LIN {X 0,Y 509.786,Z 242.479,A -85,B 0,C 180,E1 -5563.168,E2 -5563.168} C_VEL
LIN {X 0,Y 509.851,Z 242.473,A -85,B 0,C 180,E1 -5565.63,E2 -5565.63} C_VEL
LIN {X 0,Y 509.908,Z 242.464,A -85,B 0,C 180,E1 -5568.87,E2 -5568.87} C_VEL
LIN {X 0,Y 509.872,Z 242.475,A -85,B 0,C 180,E1 -5572.073,E2 -5572.073} C_VEL
LIN {X 0,Y 509.934,Z 242.462,A -85,B 0,C 180,E1 -5574.459,E2 -5574.459} C_VEL
LIN {X 0,Y 510.033,Z 242.455,A -85,B 0,C 180,E1 -5577.626,E2 -5577.626} C_VEL
LIN {X 0,Y 510.023,Z 242.454,A -85,B 0,C 180,E1 -5579.995,E2 -5579.995} C_VEL
LIN {X 0,Y 510.034,Z 242.449,A -85,B 0,C 180,E1 -5582.364,E2 -5582.364} C_VEL
LIN {X 0,Y 509.951,Z 242.467,A -85,B 0,C 180,E1 -5585.531,E2 -5585.531} C_VEL
LIN {X 0,Y 509.905,Z 242.467,A -85,B 0,C 180,E1 -5587.917,E2 -5587.917} C_VEL
LIN {X 0,Y 509.894,Z 242.471,A -85,B 0,C 180,E1 -5591.121,E2 -5591.121} C_VEL
LIN {X 0,Y 509.825,Z 242.474,A -85,B 0,C 180,E1 -5594.361,E2 -5594.361} C_VEL
LIN {X 0,Y 509.844,Z 242.475,A -85,B 0,C 180,E1 -5596.821,E2 -5596.821} C_VEL
LIN {X 0,Y 509.889,Z 242.466,A -85,B 0,C 180,E1 -5600.15,E2 -5600.15} C_VEL
LIN {X 0,Y 509.793,Z 242.48,A -85,B 0,C 180,E1 -5603.559,E2 -5603.559} C_VEL
LIN {X 0,Y 509.88,Z 242.469,A -85,B 0,C 180,E1 -5606.373,E2 -5606.373} C_VEL
LIN {X 0,Y 509.843,Z 242.481,A -85,B 0,C 180,E1 -5608.839,E2 -5608.839} C_VEL
LIN {X 0,Y 509.783,Z 242.48,A -85,B 0,C 180,E1 -5611.585,E2 -5611.585} C_VEL
LIN {X 0,Y 509.815,Z 242.48,A -85,B 0,C 180,E1 -5614.408,E2 -5614.408} C_VEL
LIN {X 0,Y 509.777,Z 242.481,A -85,B 0,C 180,E1 -5617.336,E2 -5617.336} C_VEL
LIN {X 0,Y 509.798,Z 242.485,A -85,B 0,C 180,E1 -5620.377,E2 -5620.377} C_VEL
LIN {X 0,Y 509.793,Z 242.479,A -85,B 0,C 180,E1 -5623.06,E2 -5623.06} C_VEL
LIN {X 0,Y 509.781,Z 242.482,A -85,B 0,C 180,E1 -5625.788,E2 -5625.788} C_VEL
LIN {X 0,Y 509.814,Z 242.479,A -85,B 0,C 180,E1 -5628.571,E2 -5628.571} C_VEL
LIN {X 0,Y 509.805,Z 242.479,A -85,B 0,C 180,E1 -5631.659,E2 -5631.659} C_VEL
LIN {X 0,Y 509.777,Z 242.483,A -85,B 0,C 180,E1 -5633.695,E2 -5633.695} C_VEL
LIN {X 0,Y 509.109,Z 242.568,A -85,B 0,C 180,E1 -5634.355,E2 -5634.355} C_VEL
LIN {X 0,Y 506.293,Z 242.916,A -85,B 0,C 180,E1 -5635.427,E2 -5635.427} C_VEL
LIN {X 0,Y 503.902,Z 243.217,A -85,B 0,C 180,E1 -5636.29,E2 -5636.29} C_VEL
LIN {X 0,Y 502.854,Z 243.343,A -85,B 0,C 180,E1 -5636.956,E2 -5636.956} C_VEL
LIN {X 0,Y 502.756,Z 243.355,A -85,B 0,C 180,E1 -5637.182,E2 -5637.182} C_VEL
LIN {X 0,Y 502.773,Z 243.359,A -85,B 0,C 180,E1 -5640.058,E2 -5640.058} C_VEL
LIN {X 0,Y 502.775,Z 243.353,A -85,B 0,C 180,E1 -5642.53,E2 -5642.53} C_VEL
LIN {X 0,Y 502.782,Z 243.354,A -85,B 0,C 180,E1 -5645.292,E2 -5645.292} C_VEL
LIN {X 0,Y 502.757,Z 243.361,A -85,B 0,C 180,E1 -5647.826,E2 -5647.826} C_VEL
LIN {X 0,Y 502.762,Z 243.354,A -85,B 0,C 180,E1 -5650.398,E2 -5650.398} C_VEL
LIN {X 0,Y 502.784,Z 243.355,A -85,B 0,C 180,E1 -5652.93,E2 -5652.93} C_VEL
LIN {X 0,Y 502.797,Z 243.359,A -85,B 0,C 180,E1 -5655.428,E2 -5655.428} C_VEL
LIN {X 0,Y 502.831,Z 243.349,A -85,B 0,C 180,E1 -5658.716,E2 -5658.716} C_VEL
LIN {X 0,Y 502.851,Z 243.346,A -85,B 0,C 180,E1 -5661.966,E2 -5661.966} C_VEL
LIN {X 0,Y 502.899,Z 243.34,A -85,B 0,C 180,E1 -5664.386,E2 -5664.386} C_VEL
LIN {X 0,Y 502.96,Z 243.333,A -85,B 0,C 180,E1 -5667.598,E2 -5667.598} C_VEL
LIN {X 0,Y 502.955,Z 243.333,A -85,B 0,C 180,E1 -5670,E2 -5670} C_VEL
LIN {X 0,Y 502.96,Z 243.333,A -85,B 0,C 180,E1 -5672.402,E2 -5672.402} C_VEL
LIN {X 0,Y 502.899,Z 243.34,A -85,B 0,C 180,E1 -5675.614,E2 -5675.614} C_VEL
LIN {X 0,Y 502.851,Z 243.346,A -85,B 0,C 180,E1 -5678.034,E2 -5678.034} C_VEL
LIN {X 0,Y 502.831,Z 243.349,A -85,B 0,C 180,E1 -5681.284,E2 -5681.284} C_VEL
LIN {X 0,Y 502.797,Z 243.359,A -85,B 0,C 180,E1 -5684.572,E2 -5684.572} C_VEL
LIN {X 0,Y 502.813,Z 243.352,A -85,B 0,C 180,E1 -5687.908,E2 -5687.908} C_VEL
LIN {X 0,Y 502.766,Z 243.36,A -85,B 0,C 180,E1 -5690.539,E2 -5690.539} C_VEL
LIN {X 0,Y 502.76,Z 243.355,A -85,B 0,C 180,E1 -5693.042,E2 -5693.042} C_VEL
LIN {X 0,Y 502.792,Z 243.352,A -85,B 0,C 180,E1 -5695.678,E2 -5695.678} C_VEL
LIN {X 0,Y 502.782,Z 243.357,A -85,B 0,C 180,E1 -5698.376,E2 -5698.376} C_VEL
LIN {X 0,Y 502.745,Z 243.358,A -85,B 0,C 180,E1 -5701.504,E2 -5701.504} C_VEL
LIN {X 0,Y 502.75,Z 243.358,A -85,B 0,C 180,E1 -5704.448,E2 -5704.448} C_VEL
LIN {X 0,Y 502.726,Z 243.359,A -85,B 0,C 180,E1 -5707.182,E2 -5707.182} C_VEL
LIN {X 0,Y 502.774,Z 243.358,A -85,B 0,C 180,E1 -5710.016,E2 -5710.016} C_VEL
LIN {X 0,Y 502.779,Z 243.354,A -85,B 0,C 180,E1 -5712.207,E2 -5712.207} C_VEL
LIN {X 0,Y 502.753,Z 243.361,A -85,B 0,C 180,E1 -5715.473,E2 -5715.473} C_VEL
LIN {X 0,Y 502.784,Z 243.356,A -85,B 0,C 180,E1 -5717.869,E2 -5717.869} C_VEL
LIN {X 0,Y 502.758,Z 243.357,A -85,B 0,C 180,E1 -5721.029,E2 -5721.029} C_VEL
LIN {X 0,Y 502.745,Z 243.356,A -85,B 0,C 180,E1 -5724.172,E2 -5724.172} C_VEL
LIN {X 0,Y 502.795,Z 243.354,A -85,B 0,C 180,E1 -5726.998,E2 -5726.998} C_VEL
LIN {X 0,Y 502.78,Z 243.352,A -85,B 0,C 180,E1 -5730.07,E2 -5730.07} C_VEL
LIN {X 0,Y 502.802,Z 243.35,A -85,B 0,C 180,E1 -5732.538,E2 -5732.538} C_VEL
LIN {X 0,Y 502.791,Z 243.355,A -85,B 0,C 180,E1 -5735.306,E2 -5735.306} C_VEL
LIN {X 0,Y 502.752,Z 243.355,A -85,B 0,C 180,E1 -5737.832,E2 -5737.832} C_VEL
LIN {X 0,Y 502.794,Z 243.352,A -85,B 0,C 180,E1 -5740.405,E2 -5740.405} C_VEL
LIN {X 0,Y 502.79,Z 243.358,A -85,B 0,C 180,E1 -5742.936,E2 -5742.936} C_VEL
LIN {X 0,Y 502.806,Z 243.349,A -85,B 0,C 180,E1 -5745.434,E2 -5745.434} C_VEL
LIN {X 0,Y 502.859,Z 243.35,A -85,B 0,C 180,E1 -5748.722,E2 -5748.722} C_VEL
LIN {X 0,Y 502.864,Z 243.343,A -85,B 0,C 180,E1 -5751.971,E2 -5751.971} C_VEL
LIN {X 0,Y 502.906,Z 243.344,A -85,B 0,C 180,E1 -5754.391,E2 -5754.391} C_VEL
LIN {X 0,Y 503.003,Z 243.324,A -85,B 0,C 180,E1 -5757.602,E2 -5757.602} C_VEL
LIN {X 0,Y 502.981,Z 243.329,A -85,B 0,C 180,E1 -5760.805,E2 -5760.805} C_VEL
LIN {X 0,Y 503,Z 243.331,A -85,B 0,C 180,E1 -5762.407,E2 -5762.407} C_VEL
LIN {X 0,Y 502.89,Z 243.34,A -85,B 0,C 180,E1 -5765.618,E2 -5765.618} C_VEL
LIN {X 0,Y 502.845,Z 243.352,A -85,B 0,C 180,E1 -5768.038,E2 -5768.038} C_VEL
LIN {X 0,Y 502.873,Z 243.341,A -85,B 0,C 180,E1 -5771.287,E2 -5771.287} C_VEL
LIN {X 0,Y 502.83,Z 243.346,A -85,B 0,C 180,E1 -5774.575,E2 -5774.575} C_VEL
LIN {X 0,Y 502.795,Z 243.354,A -85,B 0,C 180,E1 -5778.107,E2 -5778.107} C_VEL
LIN {X 0,Y 502.832,Z 243.345,A -85,B 0,C 180,E1 -5780.54,E2 -5780.54} C_VEL
LIN {X 0,Y 502.789,Z 243.352,A -85,B 0,C 180,E1 -5783.044,E2 -5783.044} C_VEL
LIN {X 0,Y 502.78,Z 243.358,A -85,B 0,C 180,E1 -5785.682,E2 -5785.682} C_VEL
LIN {X 0,Y 502.775,Z 243.352,A -85,B 0,C 180,E1 -5788.38,E2 -5788.38} C_VEL
LIN {X 0,Y 502.792,Z 243.355,A -85,B 0,C 180,E1 -5791.147,E2 -5791.147} C_VEL
LIN {X 0,Y 502.79,Z 243.353,A -85,B 0,C 180,E1 -5793.998,E2 -5793.998} C_VEL
LIN {X 0,Y 502.768,Z 243.362,A -85,B 0,C 180,E1 -5797.178,E2 -5797.178} C_VEL
LIN {X 0,Y 502.777,Z 243.356,A -85,B 0,C 180,E1 -5800.019,E2 -5800.019} C_VEL
LIN {X 0,Y 502.747,Z 243.365,A -85,B 0,C 180,E1 -5803.237,E2 -5803.237} C_VEL
LIN {X 0,Y 502.898,Z 244.073,A -85,B 0,C 180,E1 -5804.544,E2 -5804.544} C_VEL
LIN {X 0,Y 503.469,Z 248.342,A -85,B 0,C 180,E1 -5807.72,E2 -5807.72} C_VEL
LIN {X 0,Y 503.575,Z 250.211,A -85,B 0,C 180,E1 -5809.01,E2 -5809.01} C_VEL
LIN {X 0,Y 503.384,Z 255.037,A -85,B 0,C 180,E1 -5812.099,E2 -5812.099} C_VEL
LIN {X 0,Y 503.107,Z 260.78,A -85,B 0,C 180,E1 -5815.509,E2 -5815.509} C_VEL
LIN {X 0,Y 502.906,Z 266.132,A -85,B 0,C 180,E1 -5818.484,E2 -5818.484} C_VEL
LIN {X 0,Y 502.773,Z 270.34,A -85,B 0,C 180,E1 -5820.71,E2 -5820.71} C_VEL
LIN {X 0,Y 502.663,Z 275.73,A -85,B 0,C 180,E1 -5823.488,E2 -5823.488} C_VEL
LIN {X 0,Y 502.496,Z 281.081,A -85,B 0,C 180,E1 -5826.072,E2 -5826.072} C_VEL
LIN {X 0,Y 502.42,Z 286.478,A -85,B 0,C 180,E1 -5828.673,E2 -5828.673} C_VEL
LIN {X 0,Y 502.312,Z 291.868,A -85,B 0,C 180,E1 -5831.229,E2 -5831.229} C_VEL
LIN {X 0,Y 502.227,Z 299.054,A -85,B 0,C 180,E1 -5834.581,E2 -5834.581} C_VEL
LIN {X 0,Y 502.218,Z 301.524,A -85,B 0,C 180,E1 -5835.721,E2 -5835.721} C_VEL
LIN {X 0,Y 504.282,Z 313.728,A -85,B 0,C 180,E1 -5836.09,E2 -5836.09} C_VEL
LIN {X 0,Y 504.634,Z 317.056,A -85,B 0,C 180,E1 -5836.202,E2 -5836.202} C_VEL
LIN {X 0,Y 504.299,Z 329.38,A -85,B 0,C 180,E1 -5836.706,E2 -5836.706} C_VEL
LIN {X 0,Y 503.949,Z 339.986,A -85,B 0,C 180,E1 -5837.279,E2 -5837.279} C_VEL
LIN {X 0,Y 503.696,Z 349.477,A -85,B 0,C 180,E1 -5837.919,E2 -5837.919} C_VEL
LIN {X 0,Y 503.438,Z 358.175,A -85,B 0,C 180,E1 -5838.628,E2 -5838.628} C_VEL
LIN {X 0,Y 503.184,Z 365.542,A -85,B 0,C 180,E1 -5839.335,E2 -5839.335} C_VEL
LIN {X 0,Y 502.938,Z 372.73,A -85,B 0,C 180,E1 -5840.144,E2 -5840.144} C_VEL
LIN {X 0,Y 502.682,Z 380.276,A -85,B 0,C 180,E1 -5841.153,E2 -5841.153} C_VEL
LIN {X 0,Y 502.476,Z 386.565,A -85,B 0,C 180,E1 -5842.162,E2 -5842.162} C_VEL
LIN {X 0,Y 502.324,Z 391.989,A -85,B 0,C 180,E1 -5843.211,E2 -5843.211} C_VEL
LIN {X 0,Y 502.253,Z 396.895,A -85,B 0,C 180,E1 -5844.379,E2 -5844.379} C_VEL
LIN {X 0,Y 502.129,Z 400.851,A -85,B 0,C 180,E1 -5845.585,E2 -5845.585} C_VEL
LIN {X 0,Y 502.123,Z 403.772,A -85,B 0,C 180,E1 -5846.791,E2 -5846.791} C_VEL
LIN {X 0,Y 502.038,Z 406.196,A -85,B 0,C 180,E1 -5848.396,E2 -5848.396} C_VEL
LIN {X 0,Y 501.992,Z 406.78,A -85,B 0,C 180,E1 -5849.198,E2 -5849.198} C_VEL
LIN {X 0,Y 501.992,Z 406.78,A -85,B 0,C 180,E1 -5850.802,E2 -5850.802} C_VEL
LIN {X 0,Y 502.038,Z 406.196,A -85,B 0,C 180,E1 -5851.604,E2 -5851.604} C_VEL
LIN {X 0,Y 502.123,Z 403.772,A -85,B 0,C 180,E1 -5853.209,E2 -5853.209} C_VEL
LIN {X 0,Y 502.129,Z 400.851,A -85,B 0,C 180,E1 -5854.415,E2 -5854.415} C_VEL
LIN {X 0,Y 502.253,Z 396.895,A -85,B 0,C 180,E1 -5855.621,E2 -5855.621} C_VEL
LIN {X 0,Y 502.324,Z 391.989,A -85,B 0,C 180,E1 -5856.789,E2 -5856.789} C_VEL
LIN {X 0,Y 502.476,Z 386.565,A -85,B 0,C 180,E1 -5857.838,E2 -5857.838} C_VEL
LIN {X 0,Y 502.682,Z 380.276,A -85,B 0,C 180,E1 -5858.847,E2 -5858.847} C_VEL
LIN {X 0,Y 502.938,Z 372.73,A -85,B 0,C 180,E1 -5859.856,E2 -5859.856} C_VEL
LIN {X 0,Y 503.243,Z 363.621,A -85,B 0,C 180,E1 -5860.867,E2 -5860.867} C_VEL
LIN {X 0,Y 503.652,Z 352.174,A -85,B 0,C 180,E1 -5861.877,E2 -5861.877} C_VEL
LIN {X 0,Y 503.845,Z 342.606,A -85,B 0,C 180,E1 -5862.559,E2 -5862.559} C_VEL
LIN {X 0,Y 504.181,Z 332.396,A -85,B 0,C 180,E1 -5863.143,E2 -5863.143} C_VEL
LIN {X 0,Y 504.452,Z 322.332,A -85,B 0,C 180,E1 -5863.597,E2 -5863.597} C_VEL
LIN {X 0,Y 504.448,Z 314.602,A -85,B 0,C 180,E1 -5863.88,E2 -5863.88} C_VEL
LIN {X 0,Y 502.539,Z 303.436,A -85,B 0,C 180,E1 -5864.227,E2 -5864.227} C_VEL
LIN {X 0,Y 502.218,Z 301.524,A -85,B 0,C 180,E1 -5864.279,E2 -5864.279} C_VEL
LIN {X 0,Y 502.246,Z 295.461,A -85,B 0,C 180,E1 -5867.089,E2 -5867.089} C_VEL
LIN {X 0,Y 502.428,Z 288.275,A -85,B 0,C 180,E1 -5870.469,E2 -5870.469} C_VEL
LIN {X 0,Y 502.478,Z 282.885,A -85,B 0,C 180,E1 -5873.055,E2 -5873.055} C_VEL
LIN {X 0,Y 502.582,Z 277.398,A -85,B 0,C 180,E1 -5875.689,E2 -5875.689} C_VEL
LIN {X 0,Y 502.708,Z 272.094,A -85,B 0,C 180,E1 -5878.38,E2 -5878.38} C_VEL
LIN {X 0,Y 502.882,Z 266.832,A -85,B 0,C 180,E1 -5881.137,E2 -5881.137} C_VEL
LIN {X 0,Y 503.056,Z 261.669,A -85,B 0,C 180,E1 -5883.974,E2 -5883.974} C_VEL
LIN {X 0,Y 503.326,Z 256.07,A -85,B 0,C 180,E1 -5887.257,E2 -5887.257} C_VEL
LIN {X 0,Y 503.509,Z 251.788,A -85,B 0,C 180,E1 -5889.945,E2 -5889.945} C_VEL
LIN {X 0,Y 503.492,Z 248.328,A -85,B 0,C 180,E1 -5892.283,E2 -5892.283} C_VEL
LIN {X 0,Y 502.899,Z 244.091,A -85,B 0,C 180,E1 -5895.456,E2 -5895.456} C_VEL
LIN {X 0,Y 502.746,Z 243.362,A -85,B 0,C 180,E1 -5896.763,E2 -5896.763} C_VEL
LIN {X 0,Y 502.776,Z 243.356,A -85,B 0,C 180,E1 -5899.981,E2 -5899.981} C_VEL
LIN {X 0,Y 502.756,Z 243.36,A -85,B 0,C 180,E1 -5903.049,E2 -5903.049} C_VEL
LIN {X 0,Y 502.79,Z 243.351,A -85,B 0,C 180,E1 -5906.002,E2 -5906.002} C_VEL
LIN {X 0,Y 502.792,Z 243.355,A -85,B 0,C 180,E1 -5908.853,E2 -5908.853} C_VEL
LIN {X 0,Y 502.774,Z 243.353,A -85,B 0,C 180,E1 -5911.718,E2 -5911.718} C_VEL
LIN {X 0,Y 502.78,Z 243.358,A -85,B 0,C 180,E1 -5914.318,E2 -5914.318} C_VEL
LIN {X 0,Y 502.804,Z 243.349,A -85,B 0,C 180,E1 -5917.295,E2 -5917.295} C_VEL
LIN {X 0,Y 502.804,Z 243.356,A -85,B 0,C 180,E1 -5920.396,E2 -5920.396} C_VEL
LIN {X 0,Y 502.748,Z 243.356,A -85,B 0,C 180,E1 -5922.925,E2 -5922.925} C_VEL
LIN {X 0,Y 502.83,Z 243.346,A -85,B 0,C 180,E1 -5925.425,E2 -5925.425} C_VEL
LIN {X 0,Y 502.873,Z 243.341,A -85,B 0,C 180,E1 -5928.713,E2 -5928.713} C_VEL
LIN {X 0,Y 502.845,Z 243.352,A -85,B 0,C 180,E1 -5931.962,E2 -5931.962} C_VEL
LIN {X 0,Y 502.89,Z 243.34,A -85,B 0,C 180,E1 -5934.382,E2 -5934.382} C_VEL
LIN {X 0,Y 503.001,Z 243.331,A -85,B 0,C 180,E1 -5937.593,E2 -5937.593} C_VEL
LIN {X 0,Y 502.992,Z 243.33,A -85,B 0,C 180,E1 -5939.995,E2 -5939.995} C_VEL
LIN {X 0,Y 503.003,Z 243.324,A -85,B 0,C 180,E1 -5942.398,E2 -5942.398} C_VEL
LIN {X 0,Y 502.906,Z 243.344,A -85,B 0,C 180,E1 -5945.609,E2 -5945.609} C_VEL
LIN {X 0,Y 502.864,Z 243.343,A -85,B 0,C 180,E1 -5948.029,E2 -5948.029} C_VEL
LIN {X 0,Y 502.859,Z 243.35,A -85,B 0,C 180,E1 -5951.278,E2 -5951.278} C_VEL
LIN {X 0,Y 502.806,Z 243.349,A -85,B 0,C 180,E1 -5954.566,E2 -5954.566} C_VEL
LIN {X 0,Y 502.79,Z 243.358,A -85,B 0,C 180,E1 -5957.064,E2 -5957.064} C_VEL
LIN {X 0,Y 502.794,Z 243.352,A -85,B 0,C 180,E1 -5959.595,E2 -5959.595} C_VEL
LIN {X 0,Y 502.775,Z 243.357,A -85,B 0,C 180,E1 -5962.697,E2 -5962.697} C_VEL
LIN {X 0,Y 502.796,Z 243.35,A -85,B 0,C 180,E1 -5965.671,E2 -5965.671} C_VEL
LIN {X 0,Y 502.807,Z 243.351,A -85,B 0,C 180,E1 -5968.367,E2 -5968.367} C_VEL
LIN {X 0,Y 502.756,Z 243.355,A -85,B 0,C 180,E1 -5971.493,E2 -5971.493} C_VEL
LIN {X 0,Y 502.767,Z 243.359,A -85,B 0,C 180,E1 -5974.439,E2 -5974.439} C_VEL
LIN {X 0,Y 502.739,Z 243.358,A -85,B 0,C 180,E1 -5977.173,E2 -5977.173} C_VEL
LIN {X 0,Y 502.746,Z 243.358,A -85,B 0,C 180,E1 -5980.01,E2 -5980.01} C_VEL
LIN {X 0,Y 502.784,Z 243.357,A -85,B 0,C 180,E1 -5982.198,E2 -5982.198} C_VEL
LIN {X 0,Y 502.751,Z 243.355,A -85,B 0,C 180,E1 -5985.464,E2 -5985.464} C_VEL
LIN {X 0,Y 502.779,Z 243.355,A -85,B 0,C 180,E1 -5987.86,E2 -5987.86} C_VEL
LIN {X 0,Y 502.768,Z 243.353,A -85,B 0,C 180,E1 -5991.022,E2 -5991.022} C_VEL
LIN {X 0,Y 502.73,Z 243.365,A -85,B 0,C 180,E1 -5994.163,E2 -5994.163} C_VEL
LIN {X 0,Y 502.756,Z 243.355,A -85,B 0,C 180,E1 -5997.182,E2 -5997.182} C_VEL
LIN {X 0,Y 502.057,Z 243.449,A -85,B 0,C 180,E1 -5997.851,E2 -5997.851} C_VEL
LIN {X 0,Y 499.199,Z 243.802,A -85,B 0,C 180,E1 -5998.937,E2 -5998.937} C_VEL
LIN {X 0,Y 496.807,Z 244.103,A -85,B 0,C 180,E1 -5999.812,E2 -5999.812} C_VEL
LIN {X 0,Y 495.786,Z 244.225,A -85,B 0,C 180,E1 -6000.488,E2 -6000.488} C_VEL
LIN {X 0,Y 495.705,Z 244.233,A -85,B 0,C 180,E1 -6000.716,E2 -6000.716} C_VEL
LIN {X 0,Y 495.745,Z 244.234,A -85,B 0,C 180,E1 -6003.93,E2 -6003.93} C_VEL
LIN {X 0,Y 495.727,Z 244.232,A -85,B 0,C 180,E1 -6007.128,E2 -6007.128} C_VEL
LIN {X 0,Y 495.714,Z 244.235,A -85,B 0,C 180,E1 -6010.108,E2 -6010.108} C_VEL
LIN {X 0,Y 495.737,Z 244.232,A -85,B 0,C 180,E1 -6012.68,E2 -6012.68} C_VEL
LIN {X 0,Y 495.75,Z 244.235,A -85,B 0,C 180,E1 -6015.216,E2 -6015.216} C_VEL
LIN {X 0,Y 495.81,Z 244.222,A -85,B 0,C 180,E1 -6018.554,E2 -6018.554} C_VEL
LIN {X 0,Y 495.82,Z 244.223,A -85,B 0,C 180,E1 -6021.851,E2 -6021.851} C_VEL
LIN {X 0,Y 495.854,Z 244.217,A -85,B 0,C 180,E1 -6024.306,E2 -6024.306} C_VEL
LIN {X 0,Y 495.93,Z 244.209,A -85,B 0,C 180,E1 -6027.563,E2 -6027.563} C_VEL
LIN {X 0,Y 495.927,Z 244.209,A -85,B 0,C 180,E1 -6030,E2 -6030} C_VEL
LIN {X 0,Y 495.93,Z 244.209,A -85,B 0,C 180,E1 -6032.437,E2 -6032.437} C_VEL
LIN {X 0,Y 495.854,Z 244.217,A -85,B 0,C 180,E1 -6035.694,E2 -6035.694} C_VEL
LIN {X 0,Y 495.82,Z 244.223,A -85,B 0,C 180,E1 -6038.149,E2 -6038.149} C_VEL
LIN {X 0,Y 495.81,Z 244.222,A -85,B 0,C 180,E1 -6041.446,E2 -6041.446} C_VEL
LIN {X 0,Y 495.75,Z 244.235,A -85,B 0,C 180,E1 -6044.784,E2 -6044.784} C_VEL
LIN {X 0,Y 495.766,Z 244.233,A -85,B 0,C 180,E1 -6048.258,E2 -6048.258} C_VEL
LIN {X 0,Y 495.703,Z 244.234,A -85,B 0,C 180,E1 -6051.63,E2 -6051.63} C_VEL
LIN {X 0,Y 495.746,Z 244.229,A -85,B 0,C 180,E1 -6054.884,E2 -6054.884} C_VEL
LIN {X 0,Y 495.76,Z 244.227,A -85,B 0,C 180,E1 -6056.977,E2 -6056.977} C_VEL
LIN {X 0,Y 495.722,Z 244.239,A -85,B 0,C 180,E1 -6060.154,E2 -6060.154} C_VEL
LIN {X 0,Y 495.736,Z 244.23,A -85,B 0,C 180,E1 -6063.248,E2 -6063.248} C_VEL
LIN {X 0,Y 495.673,Z 244.243,A -85,B 0,C 180,E1 -6066.094,E2 -6066.094} C_VEL
LIN {X 0,Y 495.725,Z 244.231,A -85,B 0,C 180,E1 -6068.775,E2 -6068.775} C_VEL
LIN {X 0,Y 495.728,Z 244.239,A -85,B 0,C 180,E1 -6071.783,E2 -6071.783} C_VEL
LIN {X 0,Y 495.701,Z 244.236,A -85,B 0,C 180,E1 -6075.144,E2 -6075.144} C_VEL
LIN {X 0,Y 495.733,Z 244.231,A -85,B 0,C 180,E1 -6078.226,E2 -6078.226} C_VEL
LIN {X 0,Y 495.707,Z 244.241,A -85,B 0,C 180,E1 -6081.413,E2 -6081.413} C_VEL
LIN {X 0,Y 495.717,Z 244.232,A -85,B 0,C 180,E1 -6084.468,E2 -6084.468} C_VEL
LIN {X 0,Y 495.73,Z 244.237,A -85,B 0,C 180,E1 -6087.411,E2 -6087.411} C_VEL
LIN {X 0,Y 495.732,Z 244.23,A -85,B 0,C 180,E1 -6090.259,E2 -6090.259} C_VEL
LIN {X 0,Y 495.792,Z 244.229,A -85,B 0,C 180,E1 -6093.256,E2 -6093.256} C_VEL
LIN {X 0,Y 495.71,Z 244.233,A -85,B 0,C 180,E1 -6095.73,E2 -6095.73} C_VEL
LIN {X 0,Y 495.714,Z 244.233,A -85,B 0,C 180,E1 -6098.376,E2 -6098.376} C_VEL
LIN {X 0,Y 495.754,Z 244.234,A -85,B 0,C 180,E1 -6100.977,E2 -6100.977} C_VEL
LIN {X 0,Y 495.802,Z 244.226,A -85,B 0,C 180,E1 -6104.554,E2 -6104.554} C_VEL
LIN {X 0,Y 495.81,Z 244.221,A -85,B 0,C 180,E1 -6107.971,E2 -6107.971} C_VEL
LIN {X 0,Y 495.815,Z 244.222,A -85,B 0,C 180,E1 -6111.035,E2 -6111.035} C_VEL
LIN {X 0,Y 495.834,Z 244.217,A -85,B 0,C 180,E1 -6113.494,E2 -6113.494} C_VEL
LIN {X 0,Y 495.803,Z 244.225,A -85,B 0,C 180,E1 -6116.755,E2 -6116.755} C_VEL
LIN {X 0,Y 495.859,Z 244.222,A -85,B 0,C 180,E1 -6118.38,E2 -6118.38} C_VEL
LIN {X 0,Y 495.933,Z 244.207,A -85,B 0,C 180,E1 -6120.817,E2 -6120.817} C_VEL
LIN {X 0,Y 495.967,Z 244.206,A -85,B 0,C 180,E1 -6122.441,E2 -6122.441} C_VEL
LIN {X 0,Y 495.848,Z 244.218,A -85,B 0,C 180,E1 -6125.698,E2 -6125.698} C_VEL
LIN {X 0,Y 495.809,Z 244.228,A -85,B 0,C 180,E1 -6128.153,E2 -6128.153} C_VEL
LIN {X 0,Y 495.848,Z 244.217,A -85,B 0,C 180,E1 -6131.449,E2 -6131.449} C_VEL
LIN {X 0,Y 495.779,Z 244.224,A -85,B 0,C 180,E1 -6134.787,E2 -6134.787} C_VEL
LIN {X 0,Y 495.773,Z 244.227,A -85,B 0,C 180,E1 -6138.238,E2 -6138.238} C_VEL
LIN {X 0,Y 495.776,Z 244.224,A -85,B 0,C 180,E1 -6140.76,E2 -6140.76} C_VEL
LIN {X 0,Y 495.741,Z 244.234,A -85,B 0,C 180,E1 -6143.391,E2 -6143.391} C_VEL
LIN {X 0,Y 495.742,Z 244.229,A -85,B 0,C 180,E1 -6146.732,E2 -6146.732} C_VEL
LIN {X 0,Y 495.761,Z 244.23,A -85,B 0,C 180,E1 -6149.75,E2 -6149.75} C_VEL
LIN {X 0,Y 495.756,Z 244.227,A -85,B 0,C 180,E1 -6152.599,E2 -6152.599} C_VEL
LIN {X 0,Y 495.745,Z 244.234,A -85,B 0,C 180,E1 -6155.541,E2 -6155.541} C_VEL
LIN {X 0,Y 495.749,Z 244.234,A -85,B 0,C 180,E1 -6158.767,E2 -6158.767} C_VEL
LIN {X 0,Y 495.731,Z 244.236,A -85,B 0,C 180,E1 -6161.787,E2 -6161.787} C_VEL
LIN {X 0,Y 495.711,Z 244.301,A -85,B 0,C 180,E1 -6163.694,E2 -6163.694} C_VEL
LIN {X 0,Y 496.196,Z 247.568,A -85,B 0,C 180,E1 -6166.252,E2 -6166.252} C_VEL
LIN {X 0,Y 496.561,Z 250.8,A -85,B 0,C 180,E1 -6168.604,E2 -6168.604} C_VEL
LIN {X 0,Y 496.462,Z 255.141,A -85,B 0,C 180,E1 -6171.475,E2 -6171.475} C_VEL
LIN {X 0,Y 496.113,Z 260.072,A -85,B 0,C 180,E1 -6174.493,E2 -6174.493} C_VEL
LIN {X 0,Y 495.927,Z 265.148,A -85,B 0,C 180,E1 -6177.418,E2 -6177.418} C_VEL
LIN {X 0,Y 495.758,Z 270.337,A -85,B 0,C 180,E1 -6180.254,E2 -6180.254} C_VEL
LIN {X 0,Y 495.616,Z 276.152,A -85,B 0,C 180,E1 -6183.302,E2 -6183.302} C_VEL
LIN {X 0,Y 495.462,Z 280.973,A -85,B 0,C 180,E1 -6185.71,E2 -6185.71} C_VEL
LIN {X 0,Y 495.375,Z 286.478,A -85,B 0,C 180,E1 -6188.355,E2 -6188.355} C_VEL
LIN {X 0,Y 495.249,Z 291.868,A -85,B 0,C 180,E1 -6190.951,E2 -6190.951} C_VEL
LIN {X 0,Y 495.143,Z 297.257,A -85,B 0,C 180,E1 -6193.509,E2 -6193.509} C_VEL
LIN {X 0,Y 495.131,Z 301.524,A -85,B 0,C 180,E1 -6195.513,E2 -6195.513} C_VEL
LIN {X 0,Y 497.257,Z 313.712,A -85,B 0,C 180,E1 -6195.889,E2 -6195.889} C_VEL
LIN {X 0,Y 497.76,Z 317.061,A -85,B 0,C 180,E1 -6196.008,E2 -6196.008} C_VEL
LIN {X 0,Y 497.392,Z 329.371,A -85,B 0,C 180,E1 -6196.518,E2 -6196.518} C_VEL
LIN {X 0,Y 497.009,Z 340.234,A -85,B 0,C 180,E1 -6197.115,E2 -6197.115} C_VEL
LIN {X 0,Y 496.712,Z 349.469,A -85,B 0,C 180,E1 -6197.747,E2 -6197.747} C_VEL
LIN {X 0,Y 496.471,Z 358.169,A -85,B 0,C 180,E1 -6198.466,E2 -6198.466} C_VEL
LIN {X 0,Y 496.196,Z 365.537,A -85,B 0,C 180,E1 -6199.183,E2 -6199.183} C_VEL
LIN {X 0,Y 495.922,Z 372.726,A -85,B 0,C 180,E1 -6200.003,E2 -6200.003} C_VEL
LIN {X 0,Y 495.617,Z 380.272,A -85,B 0,C 180,E1 -6201.026,E2 -6201.026} C_VEL
LIN {X 0,Y 495.408,Z 386.56,A -85,B 0,C 180,E1 -6202.05,E2 -6202.05} C_VEL
LIN {X 0,Y 495.255,Z 391.984,A -85,B 0,C 180,E1 -6203.113,E2 -6203.113} C_VEL
LIN {X 0,Y 495.171,Z 396.891,A -85,B 0,C 180,E1 -6204.298,E2 -6204.298} C_VEL
LIN {X 0,Y 495.03,Z 400.847,A -85,B 0,C 180,E1 -6205.522,E2 -6205.522} C_VEL
LIN {X 0,Y 495.046,Z 403.769,A -85,B 0,C 180,E1 -6206.745,E2 -6206.745} C_VEL
LIN {X 0,Y 494.964,Z 406.195,A -85,B 0,C 180,E1 -6208.373,E2 -6208.373} C_VEL
LIN {X 0,Y 494.913,Z 406.779,A -85,B 0,C 180,E1 -6209.186,E2 -6209.186} C_VEL
LIN {X 0,Y 494.913,Z 406.779,A -85,B 0,C 180,E1 -6210.814,E2 -6210.814} C_VEL
LIN {X 0,Y 494.964,Z 406.195,A -85,B 0,C 180,E1 -6211.627,E2 -6211.627} C_VEL
LIN {X 0,Y 495.046,Z 403.769,A -85,B 0,C 180,E1 -6213.255,E2 -6213.255} C_VEL
LIN {X 0,Y 495.03,Z 400.847,A -85,B 0,C 180,E1 -6214.478,E2 -6214.478} C_VEL
LIN {X 0,Y 495.171,Z 396.891,A -85,B 0,C 180,E1 -6215.702,E2 -6215.702} C_VEL
LIN {X 0,Y 495.255,Z 391.984,A -85,B 0,C 180,E1 -6216.887,E2 -6216.887} C_VEL
LIN {X 0,Y 495.408,Z 386.56,A -85,B 0,C 180,E1 -6217.95,E2 -6217.95} C_VEL
LIN {X 0,Y 495.617,Z 380.272,A -85,B 0,C 180,E1 -6218.974,E2 -6218.974} C_VEL
LIN {X 0,Y 495.922,Z 372.726,A -85,B 0,C 180,E1 -6219.997,E2 -6219.997} C_VEL
LIN {X 0,Y 496.242,Z 363.619,A -85,B 0,C 180,E1 -6221.022,E2 -6221.022} C_VEL
LIN {X 0,Y 496.692,Z 352.167,A -85,B 0,C 180,E1 -6222.046,E2 -6222.046} C_VEL
LIN {X 0,Y 496.883,Z 343.088,A -85,B 0,C 180,E1 -6222.706,E2 -6222.706} C_VEL
LIN {X 0,Y 497.247,Z 332.387,A -85,B 0,C 180,E1 -6223.33,E2 -6223.33} C_VEL
LIN {X 0,Y 497.558,Z 322.322,A -85,B 0,C 180,E1 -6223.789,E2 -6223.789} C_VEL
LIN {X 0,Y 497.537,Z 315.46,A -85,B 0,C 180,E1 -6224.051,E2 -6224.051} C_VEL
LIN {X 0,Y 495.388,Z 303.15,A -85,B 0,C 180,E1 -6224.442,E2 -6224.442} C_VEL
LIN {X 0,Y 495.131,Z 301.524,A -85,B 0,C 180,E1 -6224.487,E2 -6224.487} C_VEL
LIN {X 0,Y 495.225,Z 293.99,A -85,B 0,C 180,E1 -6228.037,E2 -6228.037} C_VEL
LIN {X 0,Y 495.346,Z 288.275,A -85,B 0,C 180,E1 -6230.775,E2 -6230.775} C_VEL
LIN {X 0,Y 495.4,Z 282.812,A -85,B 0,C 180,E1 -6233.404,E2 -6233.404} C_VEL
LIN {X 0,Y 495.544,Z 277.352,A -85,B 0,C 180,E1 -6236.081,E2 -6236.081} C_VEL
LIN {X 0,Y 495.683,Z 272.09,A -85,B 0,C 180,E1 -6238.82,E2 -6238.82} C_VEL
LIN {X 0,Y 495.874,Z 266.625,A -85,B 0,C 180,E1 -6241.744,E2 -6241.744} C_VEL
LIN {X 0,Y 496.08,Z 261.362,A -85,B 0,C 180,E1 -6244.742,E2 -6244.742} C_VEL
LIN {X 0,Y 496.328,Z 256.705,A -85,B 0,C 180,E1 -6247.534,E2 -6247.534} C_VEL
LIN {X 0,Y 496.497,Z 252.642,A -85,B 0,C 180,E1 -6250.145,E2 -6250.145} C_VEL
LIN {X 0,Y 496.451,Z 249.089,A -85,B 0,C 180,E1 -6252.594,E2 -6252.594} C_VEL
LIN {X 0,Y 495.987,Z 245.779,A -85,B 0,C 180,E1 -6255.111,E2 -6255.111} C_VEL
LIN {X 0,Y 495.711,Z 244.297,A -85,B 0,C 180,E1 -6256.306,E2 -6256.306} C_VEL
LIN {X 0,Y 495.732,Z 244.236,A -85,B 0,C 180,E1 -6259.294,E2 -6259.294} C_VEL
LIN {X 0,Y 495.733,Z 244.235,A -85,B 0,C 180,E1 -6261.404,E2 -6261.404} C_VEL
LIN {X 0,Y 495.745,Z 244.233,A -85,B 0,C 180,E1 -6264.459,E2 -6264.459} C_VEL
LIN {X 0,Y 495.756,Z 244.227,A -85,B 0,C 180,E1 -6267.401,E2 -6267.401} C_VEL
LIN {X 0,Y 495.761,Z 244.23,A -85,B 0,C 180,E1 -6270.25,E2 -6270.25} C_VEL
LIN {X 0,Y 495.742,Z 244.229,A -85,B 0,C 180,E1 -6273.268,E2 -6273.268} C_VEL
LIN {X 0,Y 495.741,Z 244.234,A -85,B 0,C 180,E1 -6276.609,E2 -6276.609} C_VEL
LIN {X 0,Y 495.781,Z 244.224,A -85,B 0,C 180,E1 -6279.321,E2 -6279.321} C_VEL
LIN {X 0,Y 495.762,Z 244.229,A -85,B 0,C 180,E1 -6281.824,E2 -6281.824} C_VEL
LIN {X 0,Y 495.779,Z 244.224,A -85,B 0,C 180,E1 -6285.213,E2 -6285.213} C_VEL
LIN {X 0,Y 495.848,Z 244.217,A -85,B 0,C 180,E1 -6288.551,E2 -6288.551} C_VEL
LIN {X 0,Y 495.809,Z 244.228,A -85,B 0,C 180,E1 -6291.847,E2 -6291.847} C_VEL
LIN {X 0,Y 495.848,Z 244.218,A -85,B 0,C 180,E1 -6294.302,E2 -6294.302} C_VEL
LIN {X 0,Y 495.968,Z 244.206,A -85,B 0,C 180,E1 -6297.559,E2 -6297.559} C_VEL
LIN {X 0,Y 495.961,Z 244.205,A -85,B 0,C 180,E1 -6299.995,E2 -6299.995} C_VEL
LIN {X 0,Y 495.972,Z 244.2,A -85,B 0,C 180,E1 -6302.432,E2 -6302.432} C_VEL
LIN {X 0,Y 495.862,Z 244.22,A -85,B 0,C 180,E1 -6305.689,E2 -6305.689} C_VEL
LIN {X 0,Y 495.82,Z 244.22,A -85,B 0,C 180,E1 -6308.144,E2 -6308.144} C_VEL
LIN {X 0,Y 495.833,Z 244.224,A -85,B 0,C 180,E1 -6311.44,E2 -6311.44} C_VEL
LIN {X 0,Y 495.757,Z 244.229,A -85,B 0,C 180,E1 -6314.778,E2 -6314.778} C_VEL
LIN {X 0,Y 495.735,Z 244.236,A -85,B 0,C 180,E1 -6317.314,E2 -6317.314} C_VEL
LIN {X 0,Y 495.742,Z 244.229,A -85,B 0,C 180,E1 -6319.885,E2 -6319.885} C_VEL
LIN {X 0,Y 495.731,Z 244.236,A -85,B 0,C 180,E1 -6322.855,E2 -6322.855} C_VEL
LIN {X 0,Y 495.753,Z 244.227,A -85,B 0,C 180,E1 -6326.063,E2 -6326.063} C_VEL
LIN {X 0,Y 495.739,Z 244.237,A -85,B 0,C 180,E1 -6328.81,E2 -6328.81} C_VEL
LIN {X 0,Y 495.718,Z 244.231,A -85,B 0,C 180,E1 -6331.72,E2 -6331.72} C_VEL
LIN {X 0,Y 495.737,Z 244.237,A -85,B 0,C 180,E1 -6334.69,E2 -6334.69} C_VEL
LIN {X 0,Y 495.689,Z 244.235,A -85,B 0,C 180,E1 -6337.557,E2 -6337.557} C_VEL
LIN {X 0,Y 495.725,Z 244.236,A -85,B 0,C 180,E1 -6340.695,E2 -6340.695} C_VEL
LIN {X 0,Y 495.687,Z 244.236,A -85,B 0,C 180,E1 -6343.691,E2 -6343.691} C_VEL
LIN {X 0,Y 495.685,Z 244.244,A -85,B 0,C 180,E1 -6346.3,E2 -6346.3} C_VEL
LIN {X 0,Y 495.729,Z 244.23,A -85,B 0,C 180,E1 -6349.297,E2 -6349.297} C_VEL
LIN {X 0,Y 495.71,Z 244.233,A -85,B 0,C 180,E1 -6351.406,E2 -6351.406} C_VEL
LIN {X 0,Y 495.702,Z 244.237,A -85,B 0,C 180,E1 -6354.459,E2 -6354.459} C_VEL
LIN {X 0,Y 495.713,Z 244.234,A -85,B 0,C 180,E1 -6357.402,E2 -6357.402} C_VEL
LIN {X 0,Y 495.705,Z 244.233,A -85,B 0,C 180,E1 -6360.716,E2 -6360.716} C_VEL
LIN {X 0,Y 495.042,Z 244.32,A -85,B 0,C 180,E1 -6361.396,E2 -6361.396} C_VEL
LIN {X 0,Y 492.186,Z 244.672,A -85,B 0,C 180,E1 -6362.498,E2 -6362.498} C_VEL
LIN {X 0,Y 489.781,Z 244.974,A -85,B 0,C 180,E1 -6363.387,E2 -6363.387} C_VEL
LIN {X 0,Y 488.764,Z 245.102,A -85,B 0,C 180,E1 -6364.074,E2 -6364.074} C_VEL
LIN {X 0,Y 488.69,Z 245.107,A -85,B 0,C 180,E1 -6364.306,E2 -6364.306} C_VEL
LIN {X 0,Y 488.688,Z 245.109,A -85,B 0,C 180,E1 -6367.152,E2 -6367.152} C_VEL
LIN {X 0,Y 488.665,Z 245.117,A -85,B 0,C 180,E1 -6369.808,E2 -6369.808} C_VEL
LIN {X 0,Y 488.684,Z 245.11,A -85,B 0,C 180,E1 -6372.422,E2 -6372.422} C_VEL
LIN {X 0,Y 488.721,Z 245.108,A -85,B 0,C 180,E1 -6374.999,E2 -6374.999} C_VEL
LIN {X 0,Y 488.767,Z 245.099,A -85,B 0,C 180,E1 -6378.387,E2 -6378.387} C_VEL
LIN {X 0,Y 488.782,Z 245.101,A -85,B 0,C 180,E1 -6381.733,E2 -6381.733} C_VEL
LIN {X 0,Y 488.811,Z 245.095,A -85,B 0,C 180,E1 -6384.224,E2 -6384.224} C_VEL
LIN {X 0,Y 488.899,Z 245.086,A -85,B 0,C 180,E1 -6387.528,E2 -6387.528} C_VEL
LIN {X 0,Y 488.898,Z 245.085,A -85,B 0,C 180,E1 -6390,E2 -6390} C_VEL
LIN {X 0,Y 488.899,Z 245.086,A -85,B 0,C 180,E1 -6392.472,E2 -6392.472} C_VEL
LIN {X 0,Y 488.811,Z 245.095,A -85,B 0,C 180,E1 -6395.776,E2 -6395.776} C_VEL
LIN {X 0,Y 488.782,Z 245.101,A -85,B 0,C 180,E1 -6398.267,E2 -6398.267} C_VEL
LIN {X 0,Y 488.767,Z 245.099,A -85,B 0,C 180,E1 -6401.613,E2 -6401.613} C_VEL
LIN {X 0,Y 488.721,Z 245.108,A -85,B 0,C 180,E1 -6405.001,E2 -6405.001} C_VEL
LIN {X 0,Y 488.702,Z 245.114,A -85,B 0,C 180,E1 -6408.444,E2 -6408.444} C_VEL
LIN {X 0,Y 488.679,Z 245.109,A -85,B 0,C 180,E1 -6411.072,E2 -6411.072} C_VEL
LIN {X 0,Y 488.656,Z 245.113,A -85,B 0,C 180,E1 -6413.747,E2 -6413.747} C_VEL
LIN {X 0,Y 488.738,Z 245.102,A -85,B 0,C 180,E1 -6416.948,E2 -6416.948} C_VEL
LIN {X 0,Y 488.665,Z 245.115,A -85,B 0,C 180,E1 -6420.369,E2 -6420.369} C_VEL
LIN {X 0,Y 488.679,Z 245.11,A -85,B 0,C 180,E1 -6423.488,E2 -6423.488} C_VEL
LIN {X 0,Y 488.634,Z 245.117,A -85,B 0,C 180,E1 -6426.36,E2 -6426.36} C_VEL
LIN {X 0,Y 488.696,Z 245.108,A -85,B 0,C 180,E1 -6429.254,E2 -6429.254} C_VEL
LIN {X 0,Y 488.685,Z 245.108,A -85,B 0,C 180,E1 -6432.525,E2 -6432.525} C_VEL
LIN {X 0,Y 488.655,Z 245.115,A -85,B 0,C 180,E1 -6435.98,E2 -6435.98} C_VEL
LIN {X 0,Y 488.676,Z 245.109,A -85,B 0,C 180,E1 -6438.591,E2 -6438.591} C_VEL
LIN {X 0,Y 488.638,Z 245.117,A -85,B 0,C 180,E1 -6441.805,E2 -6441.805} C_VEL
LIN {X 0,Y 488.689,Z 245.111,A -85,B 0,C 180,E1 -6445.057,E2 -6445.057} C_VEL
LIN {X 0,Y 488.667,Z 245.11,A -85,B 0,C 180,E1 -6448.051,E2 -6448.051} C_VEL
LIN {X 0,Y 488.69,Z 245.11,A -85,B 0,C 180,E1 -6450.735,E2 -6450.735} C_VEL
LIN {X 0,Y 488.723,Z 245.106,A -85,B 0,C 180,E1 -6453.533,E2 -6453.533} C_VEL
LIN {X 0,Y 488.653,Z 245.112,A -85,B 0,C 180,E1 -6456.259,E2 -6456.259} C_VEL
LIN {X 0,Y 488.721,Z 245.108,A -85,B 0,C 180,E1 -6459.181,E2 -6459.181} C_VEL
LIN {X 0,Y 488.724,Z 245.103,A -85,B 0,C 180,E1 -6461.637,E2 -6461.637} C_VEL
LIN {X 0,Y 488.733,Z 245.107,A -85,B 0,C 180,E1 -6465.005,E2 -6465.005} C_VEL
LIN {X 0,Y 488.787,Z 245.1,A -85,B 0,C 180,E1 -6468.393,E2 -6468.393} C_VEL
LIN {X 0,Y 488.768,Z 245.097,A -85,B 0,C 180,E1 -6471.738,E2 -6471.738} C_VEL
LIN {X 0,Y 488.821,Z 245.095,A -85,B 0,C 180,E1 -6474.229,E2 -6474.229} C_VEL
LIN {X 0,Y 488.939,Z 245.076,A -85,B 0,C 180,E1 -6477.533,E2 -6477.533} C_VEL
LIN {X 0,Y 488.885,Z 245.085,A -85,B 0,C 180,E1 -6480.828,E2 -6480.828} C_VEL
LIN {X 0,Y 488.934,Z 245.082,A -85,B 0,C 180,E1 -6482.476,E2 -6482.476} C_VEL
LIN {X 0,Y 488.808,Z 245.096,A -85,B 0,C 180,E1 -6485.781,E2 -6485.781} C_VEL
LIN {X 0,Y 488.757,Z 245.104,A -85,B 0,C 180,E1 -6488.272,E2 -6488.272} C_VEL
LIN {X 0,Y 488.803,Z 245.097,A -85,B 0,C 180,E1 -6491.617,E2 -6491.617} C_VEL
LIN {X 0,Y 488.749,Z 245.1,A -85,B 0,C 180,E1 -6495.005,E2 -6495.005} C_VEL
LIN {X 0,Y 488.745,Z 245.101,A -85,B 0,C 180,E1 -6498.446,E2 -6498.446} C_VEL
LIN {X 0,Y 488.708,Z 245.106,A -85,B 0,C 180,E1 -6501.074,E2 -6501.074} C_VEL
LIN {X 0,Y 488.672,Z 245.116,A -85,B 0,C 180,E1 -6503.75,E2 -6503.75} C_VEL
LIN {X 0,Y 488.701,Z 245.107,A -85,B 0,C 180,E1 -6506.924,E2 -6506.924} C_VEL
LIN {X 0,Y 488.721,Z 245.103,A -85,B 0,C 180,E1 -6510.223,E2 -6510.223} C_VEL
LIN {X 0,Y 488.715,Z 245.111,A -85,B 0,C 180,E1 -6513.482,E2 -6513.482} C_VEL
LIN {X 0,Y 488.675,Z 245.112,A -85,B 0,C 180,E1 -6516.355,E2 -6516.355} C_VEL
LIN {X 0,Y 488.695,Z 245.115,A -85,B 0,C 180,E1 -6519.258,E2 -6519.258} C_VEL
LIN {X 0,Y 488.675,Z 245.116,A -85,B 0,C 180,E1 -6521.597,E2 -6521.597} C_VEL
LIN {X 0,Y 488.658,Z 245.118,A -85,B 0,C 180,E1 -6522.821,E2 -6522.821} C_VEL
LIN {X 0,Y 488.821,Z 245.979,A -85,B 0,C 180,E1 -6524.04,E2 -6524.04} C_VEL
LIN {X 0,Y 489.396,Z 249.888,A -85,B 0,C 180,E1 -6527.09,E2 -6527.09} C_VEL
LIN {X 0,Y 489.555,Z 252.073,A -85,B 0,C 180,E1 -6528.673,E2 -6528.673} C_VEL
LIN {X 0,Y 489.377,Z 256.881,A -85,B 0,C 180,E1 -6531.865,E2 -6531.865} C_VEL
LIN {X 0,Y 489.079,Z 261.947,A -85,B 0,C 180,E1 -6534.996,E2 -6534.996} C_VEL
LIN {X 0,Y 488.851,Z 267.193,A -85,B 0,C 180,E1 -6538.022,E2 -6538.022} C_VEL
LIN {X 0,Y 488.652,Z 272.093,A -85,B 0,C 180,E1 -6540.726,E2 -6540.726} C_VEL
LIN {X 0,Y 488.534,Z 277.349,A -85,B 0,C 180,E1 -6543.516,E2 -6543.516} C_VEL
LIN {X 0,Y 488.364,Z 282.704,A -85,B 0,C 180,E1 -6546.238,E2 -6546.238} C_VEL
LIN {X 0,Y 488.288,Z 289.07,A -85,B 0,C 180,E1 -6549.322,E2 -6549.322} C_VEL
LIN {X 0,Y 488.128,Z 295.461,A -85,B 0,C 180,E1 -6552.401,E2 -6552.401} C_VEL
LIN {X 0,Y 488.042,Z 301.524,A -85,B 0,C 180,E1 -6555.297,E2 -6555.297} C_VEL
LIN {X 0,Y 490.133,Z 313.259,A -85,B 0,C 180,E1 -6555.666,E2 -6555.666} C_VEL
LIN {X 0,Y 490.826,Z 318.453,A -85,B 0,C 180,E1 -6555.859,E2 -6555.859} C_VEL
LIN {X 0,Y 490.437,Z 330.367,A -85,B 0,C 180,E1 -6556.376,E2 -6556.376} C_VEL
LIN {X 0,Y 490.066,Z 340.486,A -85,B 0,C 180,E1 -6556.946,E2 -6556.946} C_VEL
LIN {X 0,Y 489.747,Z 349.462,A -85,B 0,C 180,E1 -6557.57,E2 -6557.57} C_VEL
LIN {X 0,Y 489.506,Z 358.163,A -85,B 0,C 180,E1 -6558.3,E2 -6558.3} C_VEL
LIN {X 0,Y 489.203,Z 365.531,A -85,B 0,C 180,E1 -6559.027,E2 -6559.027} C_VEL
LIN {X 0,Y 488.885,Z 372.721,A -85,B 0,C 180,E1 -6559.857,E2 -6559.857} C_VEL
LIN {X 0,Y 488.587,Z 380.267,A -85,B 0,C 180,E1 -6560.896,E2 -6560.896} C_VEL
LIN {X 0,Y 488.356,Z 386.556,A -85,B 0,C 180,E1 -6561.934,E2 -6561.934} C_VEL
LIN {X 0,Y 488.184,Z 391.789,A -85,B 0,C 180,E1 -6562.971,E2 -6562.971} C_VEL
LIN {X 0,Y 488.091,Z 396.886,A -85,B 0,C 180,E1 -6564.215,E2 -6564.215} C_VEL
LIN {X 0,Y 487.94,Z 400.843,A -85,B 0,C 180,E1 -6565.456,E2 -6565.456} C_VEL
LIN {X 0,Y 487.97,Z 403.767,A -85,B 0,C 180,E1 -6566.697,E2 -6566.697} C_VEL
LIN {X 0,Y 487.892,Z 406.193,A -85,B 0,C 180,E1 -6568.349,E2 -6568.349} C_VEL
LIN {X 0,Y 487.836,Z 406.777,A -85,B 0,C 180,E1 -6569.175,E2 -6569.175} C_VEL
LIN {X 0,Y 487.836,Z 406.777,A -85,B 0,C 180,E1 -6570.825,E2 -6570.825} C_VEL
LIN {X 0,Y 487.892,Z 406.193,A -85,B 0,C 180,E1 -6571.651,E2 -6571.651} C_VEL
LIN {X 0,Y 487.97,Z 403.767,A -85,B 0,C 180,E1 -6573.303,E2 -6573.303} C_VEL
LIN {X 0,Y 487.94,Z 400.843,A -85,B 0,C 180,E1 -6574.544,E2 -6574.544} C_VEL
LIN {X 0,Y 488.091,Z 396.886,A -85,B 0,C 180,E1 -6575.785,E2 -6575.785} C_VEL
LIN {X 0,Y 488.184,Z 391.789,A -85,B 0,C 180,E1 -6577.029,E2 -6577.029} C_VEL
LIN {X 0,Y 488.356,Z 386.556,A -85,B 0,C 180,E1 -6578.066,E2 -6578.066} C_VEL
LIN {X 0,Y 488.587,Z 380.267,A -85,B 0,C 180,E1 -6579.104,E2 -6579.104} C_VEL
LIN {X 0,Y 488.885,Z 372.721,A -85,B 0,C 180,E1 -6580.143,E2 -6580.143} C_VEL
LIN {X 0,Y 489.252,Z 363.616,A -85,B 0,C 180,E1 -6581.182,E2 -6581.182} C_VEL
LIN {X 0,Y 489.723,Z 352.159,A -85,B 0,C 180,E1 -6582.22,E2 -6582.22} C_VEL
LIN {X 0,Y 490.007,Z 342.005,A -85,B 0,C 180,E1 -6582.957,E2 -6582.957} C_VEL
LIN {X 0,Y 490.343,Z 332.378,A -85,B 0,C 180,E1 -6583.521,E2 -6583.521} C_VEL
LIN {X 0,Y 490.681,Z 322.313,A -85,B 0,C 180,E1 -6583.987,E2 -6583.987} C_VEL
LIN {X 0,Y 490.628,Z 316.296,A -85,B 0,C 180,E1 -6584.226,E2 -6584.226} C_VEL
LIN {X 0,Y 488.433,Z 303.714,A -85,B 0,C 180,E1 -6584.64,E2 -6584.64} C_VEL
LIN {X 0,Y 488.042,Z 301.524,A -85,B 0,C 180,E1 -6584.703,E2 -6584.703} C_VEL
LIN {X 0,Y 488.151,Z 294.315,A -85,B 0,C 180,E1 -6588.151,E2 -6588.151} C_VEL
LIN {X 0,Y 488.279,Z 288.215,A -85,B 0,C 180,E1 -6591.09,E2 -6591.09} C_VEL
LIN {X 0,Y 488.366,Z 282.704,A -85,B 0,C 180,E1 -6593.762,E2 -6593.762} C_VEL
LIN {X 0,Y 488.557,Z 276.584,A -85,B 0,C 180,E1 -6596.885,E2 -6596.885} C_VEL
LIN {X 0,Y 488.744,Z 270.066,A -85,B 0,C 180,E1 -6600.366,E2 -6600.366} C_VEL
LIN {X 0,Y 488.951,Z 264.465,A -85,B 0,C 180,E1 -6603.519,E2 -6603.519} C_VEL
LIN {X 0,Y 489.175,Z 259.589,A -85,B 0,C 180,E1 -6606.429,E2 -6606.429} C_VEL
LIN {X 0,Y 489.446,Z 255.239,A -85,B 0,C 180,E1 -6609.182,E2 -6609.182} C_VEL
LIN {X 0,Y 489.543,Z 251.52,A -85,B 0,C 180,E1 -6611.707,E2 -6611.707} C_VEL
LIN {X 0,Y 489.177,Z 248.329,A -85,B 0,C 180,E1 -6614.078,E2 -6614.078} C_VEL
LIN {X 0,Y 488.73,Z 245.513,A -85,B 0,C 180,E1 -6616.347,E2 -6616.347} C_VEL
LIN {X 0,Y 488.655,Z 245.117,A -85,B 0,C 180,E1 -6617.467,E2 -6617.467} C_VEL
LIN {X 0,Y 488.711,Z 245.109,A -85,B 0,C 180,E1 -6619.671,E2 -6619.671} C_VEL
LIN {X 0,Y 488.671,Z 245.118,A -85,B 0,C 180,E1 -6622.837,E2 -6622.837} C_VEL
LIN {X 0,Y 488.723,Z 245.103,A -85,B 0,C 180,E1 -6625.883,E2 -6625.883} C_VEL
LIN {X 0,Y 488.691,Z 245.112,A -85,B 0,C 180,E1 -6628.817,E2 -6628.817} C_VEL
LIN {X 0,Y 488.697,Z 245.106,A -85,B 0,C 180,E1 -6631.665,E2 -6631.665} C_VEL
LIN {X 0,Y 488.702,Z 245.107,A -85,B 0,C 180,E1 -6634.956,E2 -6634.956} C_VEL
LIN {X 0,Y 488.697,Z 245.11,A -85,B 0,C 180,E1 -6638.039,E2 -6638.039} C_VEL
LIN {X 0,Y 488.728,Z 245.105,A -85,B 0,C 180,E1 -6640.682,E2 -6640.682} C_VEL
LIN {X 0,Y 488.671,Z 245.109,A -85,B 0,C 180,E1 -6643.279,E2 -6643.279} C_VEL
LIN {X 0,Y 488.726,Z 245.107,A -85,B 0,C 180,E1 -6645.846,E2 -6645.846} C_VEL
LIN {X 0,Y 488.803,Z 245.097,A -85,B 0,C 180,E1 -6648.383,E2 -6648.383} C_VEL
LIN {X 0,Y 488.757,Z 245.104,A -85,B 0,C 180,E1 -6651.728,E2 -6651.728} C_VEL
LIN {X 0,Y 488.808,Z 245.096,A -85,B 0,C 180,E1 -6654.219,E2 -6654.219} C_VEL
LIN {X 0,Y 488.934,Z 245.082,A -85,B 0,C 180,E1 -6657.524,E2 -6657.524} C_VEL
LIN {X 0,Y 488.931,Z 245.081,A -85,B 0,C 180,E1 -6659.995,E2 -6659.995} C_VEL
LIN {X 0,Y 488.939,Z 245.076,A -85,B 0,C 180,E1 -6662.467,E2 -6662.467} C_VEL
LIN {X 0,Y 488.821,Z 245.095,A -85,B 0,C 180,E1 -6665.771,E2 -6665.771} C_VEL
LIN {X 0,Y 488.768,Z 245.097,A -85,B 0,C 180,E1 -6668.262,E2 -6668.262} C_VEL
LIN {X 0,Y 488.787,Z 245.1,A -85,B 0,C 180,E1 -6671.607,E2 -6671.607} C_VEL
LIN {X 0,Y 488.733,Z 245.107,A -85,B 0,C 180,E1 -6674.995,E2 -6674.995} C_VEL
LIN {X 0,Y 488.722,Z 245.104,A -85,B 0,C 180,E1 -6678.437,E2 -6678.437} C_VEL
LIN {X 0,Y 488.68,Z 245.117,A -85,B 0,C 180,E1 -6681.065,E2 -6681.065} C_VEL
LIN {X 0,Y 488.653,Z 245.112,A -85,B 0,C 180,E1 -6683.741,E2 -6683.741} C_VEL
LIN {X 0,Y 488.761,Z 245.106,A -85,B 0,C 180,E1 -6686.938,E2 -6686.938} C_VEL
LIN {X 0,Y 488.674,Z 245.112,A -85,B 0,C 180,E1 -6690.357,E2 -6690.357} C_VEL
LIN {X 0,Y 488.698,Z 245.106,A -85,B 0,C 180,E1 -6693.479,E2 -6693.479} C_VEL
LIN {X 0,Y 488.648,Z 245.117,A -85,B 0,C 180,E1 -6696.35,E2 -6696.35} C_VEL
LIN {X 0,Y 488.658,Z 245.112,A -85,B 0,C 180,E1 -6699.249,E2 -6699.249} C_VEL
LIN {X 0,Y 488.689,Z 245.114,A -85,B 0,C 180,E1 -6702.516,E2 -6702.516} C_VEL
LIN {X 0,Y 488.653,Z 245.115,A -85,B 0,C 180,E1 -6705.971,E2 -6705.971} C_VEL
LIN {X 0,Y 488.672,Z 245.113,A -85,B 0,C 180,E1 -6708.582,E2 -6708.582} C_VEL
LIN {X 0,Y 488.694,Z 245.107,A -85,B 0,C 180,E1 -6710.937,E2 -6710.937} C_VEL
LIN {X 0,Y 488.63,Z 245.12,A -85,B 0,C 180,E1 -6713.865,E2 -6713.865} C_VEL
LIN {X 0,Y 488.682,Z 245.108,A -85,B 0,C 180,E1 -6716.874,E2 -6716.874} C_VEL
LIN {X 0,Y 488.679,Z 245.115,A -85,B 0,C 180,E1 -6719.778,E2 -6719.778} C_VEL
LIN {X 0,Y 488.738,Z 245.102,A -85,B 0,C 180,E1 -6723.052,E2 -6723.052} C_VEL
LIN {X 0,Y 488.69,Z 245.107,A -85,B 0,C 180,E1 -6724.306,E2 -6724.306} C_VEL
LIN {X 0,Y 488.044,Z 245.191,A -85,B 0,C 180,E1 -6724.994,E2 -6724.994} C_VEL
LIN {X 0,Y 485.183,Z 245.554,A -85,B 0,C 180,E1 -6726.11,E2 -6726.11} C_VEL
LIN {X 0,Y 482.744,Z 245.859,A -85,B 0,C 180,E1 -6727.01,E2 -6727.01} C_VEL
LIN {X 0,Y 481.69,Z 245.987,A -85,B 0,C 180,E1 -6727.706,E2 -6727.706} C_VEL
LIN {X 0,Y 481.602,Z 245.994,A -85,B 0,C 180,E1 -6727.941,E2 -6727.941} C_VEL
LIN {X 0,Y 481.644,Z 245.985,A -85,B 0,C 180,E1 -6730.391,E2 -6730.391} C_VEL
LIN {X 0,Y 481.638,Z 245.99,A -85,B 0,C 180,E1 -6733.032,E2 -6733.032} C_VEL
LIN {X 0,Y 481.644,Z 245.991,A -85,B 0,C 180,E1 -6735.638,E2 -6735.638} C_VEL
LIN {X 0,Y 481.73,Z 245.976,A -85,B 0,C 180,E1 -6738.215,E2 -6738.215} C_VEL
LIN {X 0,Y 481.724,Z 245.98,A -85,B 0,C 180,E1 -6741.611,E2 -6741.611} C_VEL
LIN {X 0,Y 481.771,Z 245.972,A -85,B 0,C 180,E1 -6744.139,E2 -6744.139} C_VEL
LIN {X 0,Y 481.867,Z 245.962,A -85,B 0,C 180,E1 -6747.492,E2 -6747.492} C_VEL
LIN {X 0,Y 481.87,Z 245.96,A -85,B 0,C 180,E1 -6750,E2 -6750} C_VEL
LIN {X 0,Y 481.867,Z 245.962,A -85,B 0,C 180,E1 -6752.508,E2 -6752.508} C_VEL
LIN {X 0,Y 481.771,Z 245.972,A -85,B 0,C 180,E1 -6755.861,E2 -6755.861} C_VEL
LIN {X 0,Y 481.724,Z 245.98,A -85,B 0,C 180,E1 -6758.389,E2 -6758.389} C_VEL
LIN {X 0,Y 481.73,Z 245.976,A -85,B 0,C 180,E1 -6761.785,E2 -6761.785} C_VEL
LIN {X 0,Y 481.698,Z 245.982,A -85,B 0,C 180,E1 -6765.225,E2 -6765.225} C_VEL
LIN {X 0,Y 481.653,Z 245.99,A -85,B 0,C 180,E1 -6768.724,E2 -6768.724} C_VEL
LIN {X 0,Y 481.614,Z 245.988,A -85,B 0,C 180,E1 -6771.396,E2 -6771.396} C_VEL
LIN {X 0,Y 481.637,Z 245.992,A -85,B 0,C 180,E1 -6774.115,E2 -6774.115} C_VEL
LIN {X 0,Y 481.691,Z 245.979,A -85,B 0,C 180,E1 -6777.144,E2 -6777.144} C_VEL
LIN {X 0,Y 481.631,Z 245.99,A -85,B 0,C 180,E1 -6779.744,E2 -6779.744} C_VEL
LIN {X 0,Y 481.617,Z 245.989,A -85,B 0,C 180,E1 -6782.678,E2 -6782.678} C_VEL
LIN {X 0,Y 481.587,Z 245.997,A -85,B 0,C 180,E1 -6785.713,E2 -6785.713} C_VEL
LIN {X 0,Y 481.667,Z 245.984,A -85,B 0,C 180,E1 -6789.359,E2 -6789.359} C_VEL
LIN {X 0,Y 481.624,Z 245.99,A -85,B 0,C 180,E1 -6792.162,E2 -6792.162} C_VEL
LIN {X 0,Y 481.612,Z 245.989,A -85,B 0,C 180,E1 -6794.462,E2 -6794.462} C_VEL
LIN {X 0,Y 481.643,Z 245.985,A -85,B 0,C 180,E1 -6796.851,E2 -6796.851} C_VEL
LIN {X 0,Y 481.633,Z 245.988,A -85,B 0,C 180,E1 -6800.065,E2 -6800.065} C_VEL
LIN {X 0,Y 481.588,Z 245.998,A -85,B 0,C 180,E1 -6803.258,E2 -6803.258} C_VEL
LIN {X 0,Y 481.672,Z 245.981,A -85,B 0,C 180,E1 -6806.335,E2 -6806.335} C_VEL
LIN {X 0,Y 481.615,Z 245.994,A -85,B 0,C 180,E1 -6809.423,E2 -6809.423} C_VEL
LIN {X 0,Y 481.668,Z 245.982,A -85,B 0,C 180,E1 -6812.173,E2 -6812.173} C_VEL
LIN {X 0,Y 481.677,Z 245.988,A -85,B 0,C 180,E1 -6814.975,E2 -6814.975} C_VEL
LIN {X 0,Y 481.62,Z 245.988,A -85,B 0,C 180,E1 -6817.71,E2 -6817.71} C_VEL
LIN {X 0,Y 481.677,Z 245.983,A -85,B 0,C 180,E1 -6820.398,E2 -6820.398} C_VEL
LIN {X 0,Y 481.652,Z 245.989,A -85,B 0,C 180,E1 -6823.039,E2 -6823.039} C_VEL
LIN {X 0,Y 481.656,Z 245.983,A -85,B 0,C 180,E1 -6825.644,E2 -6825.644} C_VEL
LIN {X 0,Y 481.733,Z 245.976,A -85,B 0,C 180,E1 -6828.22,E2 -6828.22} C_VEL
LIN {X 0,Y 481.723,Z 245.975,A -85,B 0,C 180,E1 -6831.616,E2 -6831.616} C_VEL
LIN {X 0,Y 481.783,Z 245.971,A -85,B 0,C 180,E1 -6834.144,E2 -6834.144} C_VEL
LIN {X 0,Y 481.906,Z 245.952,A -85,B 0,C 180,E1 -6837.497,E2 -6837.497} C_VEL
LIN {X 0,Y 481.838,Z 245.962,A -85,B 0,C 180,E1 -6840.841,E2 -6840.841} C_VEL
LIN {X 0,Y 481.899,Z 245.957,A -85,B 0,C 180,E1 -6842.512,E2 -6842.512} C_VEL
LIN {X 0,Y 481.769,Z 245.974,A -85,B 0,C 180,E1 -6845.866,E2 -6845.866} C_VEL
LIN {X 0,Y 481.716,Z 245.98,A -85,B 0,C 180,E1 -6848.393,E2 -6848.393} C_VEL
LIN {X 0,Y 481.749,Z 245.978,A -85,B 0,C 180,E1 -6851.789,E2 -6851.789} C_VEL
LIN {X 0,Y 481.73,Z 245.975,A -85,B 0,C 180,E1 -6855.229,E2 -6855.229} C_VEL
LIN {X 0,Y 481.705,Z 245.977,A -85,B 0,C 180,E1 -6858.726,E2 -6858.726} C_VEL
LIN {X 0,Y 481.646,Z 245.989,A -85,B 0,C 180,E1 -6861.399,E2 -6861.399} C_VEL
LIN {X 0,Y 481.651,Z 245.986,A -85,B 0,C 180,E1 -6864.118,E2 -6864.118} C_VEL
LIN {X 0,Y 481.656,Z 245.987,A -85,B 0,C 180,E1 -6867.12,E2 -6867.12} C_VEL
LIN {X 0,Y 481.67,Z 245.986,A -85,B 0,C 180,E1 -6869.745,E2 -6869.745} C_VEL
LIN {X 0,Y 481.657,Z 245.984,A -85,B 0,C 180,E1 -6872.679,E2 -6872.679} C_VEL
LIN {X 0,Y 481.634,Z 245.991,A -85,B 0,C 180,E1 -6875.713,E2 -6875.713} C_VEL
LIN {X 0,Y 481.664,Z 245.99,A -85,B 0,C 180,E1 -6878.863,E2 -6878.863} C_VEL
LIN {X 0,Y 481.628,Z 245.993,A -85,B 0,C 180,E1 -6881.911,E2 -6881.911} C_VEL
LIN {X 0,Y 481.67,Z 246.353,A -85,B 0,C 180,E1 -6883.3,E2 -6883.3} C_VEL
LIN {X 0,Y 482.222,Z 249.879,A -85,B 0,C 180,E1 -6886.175,E2 -6886.175} C_VEL
LIN {X 0,Y 482.493,Z 252.287,A -85,B 0,C 180,E1 -6887.98,E2 -6887.98} C_VEL
LIN {X 0,Y 482.445,Z 255.954,A -85,B 0,C 180,E1 -6890.544,E2 -6890.544} C_VEL
LIN {X 0,Y 482.296,Z 258.587,A -85,B 0,C 180,E1 -6892.265,E2 -6892.265} C_VEL
LIN {X 0,Y 482.015,Z 263.554,A -85,B 0,C 180,E1 -6895.345,E2 -6895.345} C_VEL
LIN {X 0,Y 481.773,Z 268.628,A -85,B 0,C 180,E1 -6898.322,E2 -6898.322} C_VEL
LIN {X 0,Y 481.582,Z 273.836,A -85,B 0,C 180,E1 -6901.211,E2 -6901.211} C_VEL
LIN {X 0,Y 481.434,Z 279.1,A -85,B 0,C 180,E1 -6904.028,E2 -6904.028} C_VEL
LIN {X 0,Y 481.281,Z 284.73,A -85,B 0,C 180,E1 -6906.926,E2 -6906.926} C_VEL
LIN {X 0,Y 481.193,Z 289.942,A -85,B 0,C 180,E1 -6909.481,E2 -6909.481} C_VEL
LIN {X 0,Y 481.052,Z 295.433,A -85,B 0,C 180,E1 -6912.134,E2 -6912.134} C_VEL
LIN {X 0,Y 481.002,Z 301.524,A -85,B 0,C 180,E1 -6915.077,E2 -6915.077} C_VEL
LIN {X 0,Y 483.071,Z 313.109,A -85,B 0,C 180,E1 -6915.448,E2 -6915.448} C_VEL
LIN {X 0,Y 483.878,Z 319.731,A -85,B 0,C 180,E1 -6915.705,E2 -6915.705} C_VEL
LIN {X 0,Y 483.538,Z 330.358,A -85,B 0,C 180,E1 -6916.178,E2 -6916.178} C_VEL
LIN {X 0,Y 483.145,Z 340.805,A -85,B 0,C 180,E1 -6916.777,E2 -6916.777} C_VEL
LIN {X 0,Y 482.794,Z 349.454,A -85,B 0,C 180,E1 -6917.388,E2 -6917.388} C_VEL
LIN {X 0,Y 482.538,Z 358.156,A -85,B 0,C 180,E1 -6918.128,E2 -6918.128} C_VEL
LIN {X 0,Y 482.194,Z 365.526,A -85,B 0,C 180,E1 -6918.865,E2 -6918.865} C_VEL
LIN {X 0,Y 481.88,Z 372.717,A -85,B 0,C 180,E1 -6919.708,E2 -6919.708} C_VEL
LIN {X 0,Y 481.557,Z 380.263,A -85,B 0,C 180,E1 -6920.762,E2 -6920.762} C_VEL
LIN {X 0,Y 481.322,Z 386.551,A -85,B 0,C 180,E1 -6921.815,E2 -6921.815} C_VEL
LIN {X 0,Y 481.105,Z 391.784,A -85,B 0,C 180,E1 -6922.867,E2 -6922.867} C_VEL
LIN {X 0,Y 480.989,Z 395.564,A -85,B 0,C 180,E1 -6923.77,E2 -6923.77} C_VEL
LIN {X 0,Y 480.908,Z 399.632,A -85,B 0,C 180,E1 -6924.97,E2 -6924.97} C_VEL
LIN {X 0,Y 480.849,Z 401.975,A -85,B 0,C 180,E1 -6925.809,E2 -6925.809} C_VEL
LIN {X 0,Y 480.895,Z 403.763,A -85,B 0,C 180,E1 -6926.649,E2 -6926.649} C_VEL
LIN {X 0,Y 480.793,Z 406.19,A -85,B 0,C 180,E1 -6928.325,E2 -6928.325} C_VEL
LIN {X 0,Y 480.763,Z 406.773,A -85,B 0,C 180,E1 -6929.162,E2 -6929.162} C_VEL
LIN {X 0,Y 480.763,Z 406.773,A -85,B 0,C 180,E1 -6930.838,E2 -6930.838} C_VEL
LIN {X 0,Y 480.793,Z 406.19,A -85,B 0,C 180,E1 -6931.675,E2 -6931.675} C_VEL
LIN {X 0,Y 480.895,Z 403.763,A -85,B 0,C 180,E1 -6933.351,E2 -6933.351} C_VEL
LIN {X 0,Y 480.856,Z 400.84,A -85,B 0,C 180,E1 -6934.611,E2 -6934.611} C_VEL
LIN {X 0,Y 481.01,Z 396.882,A -85,B 0,C 180,E1 -6935.87,E2 -6935.87} C_VEL
LIN {X 0,Y 481.068,Z 393.686,A -85,B 0,C 180,E1 -6936.712,E2 -6936.712} C_VEL
LIN {X 0,Y 481.252,Z 387.701,A -85,B 0,C 180,E1 -6937.974,E2 -6937.974} C_VEL
LIN {X 0,Y 481.519,Z 381.633,A -85,B 0,C 180,E1 -6939.027,E2 -6939.027} C_VEL
LIN {X 0,Y 481.826,Z 374.338,A -85,B 0,C 180,E1 -6940.08,E2 -6940.08} C_VEL
LIN {X 0,Y 482.07,Z 367.439,A -85,B 0,C 180,E1 -6940.925,E2 -6940.925} C_VEL
LIN {X 0,Y 482.466,Z 359.288,A -85,B 0,C 180,E1 -6941.767,E2 -6941.767} C_VEL
LIN {X 0,Y 482.78,Z 350.802,A -85,B 0,C 180,E1 -6942.506,E2 -6942.506} C_VEL
LIN {X 0,Y 483.068,Z 342.596,A -85,B 0,C 180,E1 -6943.107,E2 -6943.107} C_VEL
LIN {X 0,Y 483.45,Z 332.369,A -85,B 0,C 180,E1 -6943.717,E2 -6943.717} C_VEL
LIN {X 0,Y 483.789,Z 322.303,A -85,B 0,C 180,E1 -6944.19,E2 -6944.19} C_VEL
LIN {X 0,Y 483.689,Z 317.071,A -85,B 0,C 180,E1 -6944.408,E2 -6944.408} C_VEL
LIN {X 0,Y 481.406,Z 303.836,A -85,B 0,C 180,E1 -6944.856,E2 -6944.856} C_VEL
LIN {X 0,Y 481.002,Z 301.524,A -85,B 0,C 180,E1 -6944.923,E2 -6944.923} C_VEL
LIN {X 0,Y 481.072,Z 294.602,A -85,B 0,C 180,E1 -6948.266,E2 -6948.266} C_VEL
LIN {X 0,Y 481.214,Z 288.108,A -85,B 0,C 180,E1 -6951.414,E2 -6951.414} C_VEL
LIN {X 0,Y 481.317,Z 282.608,A -85,B 0,C 180,E1 -6954.132,E2 -6954.132} C_VEL
LIN {X 0,Y 481.515,Z 276.997,A -85,B 0,C 180,E1 -6957.081,E2 -6957.081} C_VEL
LIN {X 0,Y 481.715,Z 270.536,A -85,B 0,C 180,E1 -6960.592,E2 -6960.592} C_VEL
LIN {X 0,Y 481.944,Z 265.004,A -85,B 0,C 180,E1 -6963.773,E2 -6963.773} C_VEL
LIN {X 0,Y 482.186,Z 260.193,A -85,B 0,C 180,E1 -6966.71,E2 -6966.71} C_VEL
LIN {X 0,Y 482.442,Z 255.949,A -85,B 0,C 180,E1 -6969.456,E2 -6969.456} C_VEL
LIN {X 0,Y 482.493,Z 252.189,A -85,B 0,C 180,E1 -6972.069,E2 -6972.069} C_VEL
LIN {X 0,Y 482.143,Z 249.123,A -85,B 0,C 180,E1 -6974.415,E2 -6974.415} C_VEL
LIN {X 0,Y 481.634,Z 246.166,A -85,B 0,C 180,E1 -6976.852,E2 -6976.852} C_VEL
LIN {X 0,Y 481.663,Z 245.987,A -85,B 0,C 180,E1 -6980.055,E2 -6980.055} C_VEL
LIN {X 0,Y 481.626,Z 245.989,A -85,B 0,C 180,E1 -6983.375,E2 -6983.375} C_VEL
LIN {X 0,Y 481.677,Z 245.984,A -85,B 0,C 180,E1 -6986.324,E2 -6986.324} C_VEL
LIN {X 0,Y 481.648,Z 245.985,A -85,B 0,C 180,E1 -6989.416,E2 -6989.416} C_VEL
LIN {X 0,Y 481.653,Z 245.987,A -85,B 0,C 180,E1 -6992.161,E2 -6992.161} C_VEL
LIN {X 0,Y 481.677,Z 245.983,A -85,B 0,C 180,E1 -6994.964,E2 -6994.964} C_VEL
LIN {X 0,Y 481.648,Z 245.985,A -85,B 0,C 180,E1 -6997.701,E2 -6997.701} C_VEL
LIN {X 0,Y 481.694,Z 245.985,A -85,B 0,C 180,E1 -7000.389,E2 -7000.389} C_VEL
LIN {X 0,Y 481.614,Z 245.989,A -85,B 0,C 180,E1 -7003.027,E2 -7003.027} C_VEL
LIN {X 0,Y 481.677,Z 245.983,A -85,B 0,C 180,E1 -7005.634,E2 -7005.634} C_VEL
LIN {X 0,Y 481.749,Z 245.978,A -85,B 0,C 180,E1 -7008.211,E2 -7008.211} C_VEL
LIN {X 0,Y 481.716,Z 245.98,A -85,B 0,C 180,E1 -7011.607,E2 -7011.607} C_VEL
LIN {X 0,Y 481.769,Z 245.974,A -85,B 0,C 180,E1 -7014.134,E2 -7014.134} C_VEL
LIN {X 0,Y 481.9,Z 245.957,A -85,B 0,C 180,E1 -7017.488,E2 -7017.488} C_VEL
LIN {X 0,Y 481.9,Z 245.957,A -85,B 0,C 180,E1 -7019.995,E2 -7019.995} C_VEL
LIN {X 0,Y 481.906,Z 245.952,A -85,B 0,C 180,E1 -7022.503,E2 -7022.503} C_VEL
LIN {X 0,Y 481.783,Z 245.971,A -85,B 0,C 180,E1 -7025.856,E2 -7025.856} C_VEL
LIN {X 0,Y 481.723,Z 245.975,A -85,B 0,C 180,E1 -7028.384,E2 -7028.384} C_VEL
LIN {X 0,Y 481.733,Z 245.976,A -85,B 0,C 180,E1 -7031.78,E2 -7031.78} C_VEL
LIN {X 0,Y 481.717,Z 245.984,A -85,B 0,C 180,E1 -7035.219,E2 -7035.219} C_VEL
LIN {X 0,Y 481.683,Z 245.983,A -85,B 0,C 180,E1 -7038.717,E2 -7038.717} C_VEL
LIN {X 0,Y 481.618,Z 245.992,A -85,B 0,C 180,E1 -7041.389,E2 -7041.389} C_VEL
LIN {X 0,Y 481.639,Z 245.986,A -85,B 0,C 180,E1 -7044.108,E2 -7044.108} C_VEL
LIN {X 0,Y 481.715,Z 245.981,A -85,B 0,C 180,E1 -7047.134,E2 -7047.134} C_VEL
LIN {X 0,Y 481.645,Z 245.985,A -85,B 0,C 180,E1 -7049.736,E2 -7049.736} C_VEL
LIN {X 0,Y 481.635,Z 245.994,A -85,B 0,C 180,E1 -7052.669,E2 -7052.669} C_VEL
LIN {X 0,Y 481.603,Z 245.99,A -85,B 0,C 180,E1 -7055.704,E2 -7055.704} C_VEL
LIN {X 0,Y 481.628,Z 245.991,A -85,B 0,C 180,E1 -7058.854,E2 -7058.854} C_VEL
LIN {X 0,Y 481.629,Z 245.991,A -85,B 0,C 180,E1 -7062.153,E2 -7062.153} C_VEL
LIN {X 0,Y 481.613,Z 245.996,A -85,B 0,C 180,E1 -7064.453,E2 -7064.453} C_VEL
LIN {X 0,Y 481.64,Z 245.987,A -85,B 0,C 180,E1 -7066.841,E2 -7066.841} C_VEL
LIN {X 0,Y 481.64,Z 245.992,A -85,B 0,C 180,E1 -7070.057,E2 -7070.057} C_VEL
LIN {X 0,Y 481.574,Z 245.994,A -85,B 0,C 180,E1 -7073.249,E2 -7073.249} C_VEL
LIN {X 0,Y 481.653,Z 245.988,A -85,B 0,C 180,E1 -7076.326,E2 -7076.326} C_VEL
LIN {X 0,Y 481.604,Z 245.992,A -85,B 0,C 180,E1 -7079.411,E2 -7079.411} C_VEL
LIN {X 0,Y 481.642,Z 245.989,A -85,B 0,C 180,E1 -7082.165,E2 -7082.165} C_VEL
LIN {X 0,Y 481.674,Z 245.981,A -85,B 0,C 180,E1 -7084.968,E2 -7084.968} C_VEL
LIN {X 0,Y 481.602,Z 245.994,A -85,B 0,C 180,E1 -7087.941,E2 -7087.941} C_VEL
LIN {X 0,Y 480.931,Z 246.075,A -85,B 0,C 180,E1 -7088.639,E2 -7088.639} C_VEL
LIN {X 0,Y 478.094,Z 246.434,A -85,B 0,C 180,E1 -7089.773,E2 -7089.773} C_VEL
LIN {X 0,Y 475.703,Z 246.731,A -85,B 0,C 180,E1 -7090.687,E2 -7090.687} C_VEL
LIN {X 0,Y 474.683,Z 246.858,A -85,B 0,C 180,E1 -7091.393,E2 -7091.393} C_VEL
LIN {X 0,Y 474.602,Z 246.867,A -85,B 0,C 180,E1 -7091.632,E2 -7091.632} C_VEL
LIN {X 0,Y 474.652,Z 246.859,A -85,B 0,C 180,E1 -7094.543,E2 -7094.543} C_VEL
LIN {X 0,Y 474.673,Z 246.856,A -85,B 0,C 180,E1 -7098.037,E2 -7098.037} C_VEL
LIN {X 0,Y 474.682,Z 246.858,A -85,B 0,C 180,E1 -7101.486,E2 -7101.486} C_VEL
LIN {X 0,Y 474.733,Z 246.849,A -85,B 0,C 180,E1 -7104.052,E2 -7104.052} C_VEL
LIN {X 0,Y 474.834,Z 246.839,A -85,B 0,C 180,E1 -7107.455,E2 -7107.455} C_VEL
LIN {X 0,Y 474.841,Z 246.836,A -85,B 0,C 180,E1 -7110,E2 -7110} C_VEL
LIN {X 0,Y 474.834,Z 246.839,A -85,B 0,C 180,E1 -7112.545,E2 -7112.545} C_VEL
LIN {X 0,Y 474.733,Z 246.849,A -85,B 0,C 180,E1 -7115.948,E2 -7115.948} C_VEL
LIN {X 0,Y 474.682,Z 246.858,A -85,B 0,C 180,E1 -7118.514,E2 -7118.514} C_VEL
LIN {X 0,Y 474.673,Z 246.856,A -85,B 0,C 180,E1 -7121.963,E2 -7121.963} C_VEL
LIN {X 0,Y 474.649,Z 246.86,A -85,B 0,C 180,E1 -7125.784,E2 -7125.784} C_VEL
LIN {X 0,Y 474.604,Z 246.864,A -85,B 0,C 180,E1 -7129.012,E2 -7129.012} C_VEL
LIN {X 0,Y 474.582,Z 246.866,A -85,B 0,C 180,E1 -7131.729,E2 -7131.729} C_VEL
LIN {X 0,Y 474.616,Z 246.865,A -85,B 0,C 180,E1 -7134.495,E2 -7134.495} C_VEL
LIN {X 0,Y 474.639,Z 246.858,A -85,B 0,C 180,E1 -7137.342,E2 -7137.342} C_VEL
LIN {X 0,Y 474.555,Z 246.868,A -85,B 0,C 180,E1 -7140.816,E2 -7140.816} C_VEL
LIN {X 0,Y 474.583,Z 246.873,A -85,B 0,C 180,E1 -7143.988,E2 -7143.988} C_VEL
LIN {X 0,Y 474.521,Z 246.872,A -85,B 0,C 180,E1 -7146.904,E2 -7146.904} C_VEL
LIN {X 0,Y 474.603,Z 246.868,A -85,B 0,C 180,E1 -7149.656,E2 -7149.656} C_VEL
LIN {X 0,Y 474.603,Z 246.862,A -85,B 0,C 180,E1 -7152.935,E2 -7152.935} C_VEL
LIN {X 0,Y 474.571,Z 246.87,A -85,B 0,C 180,E1 -7155.901,E2 -7155.901} C_VEL
LIN {X 0,Y 474.589,Z 246.866,A -85,B 0,C 180,E1 -7159.045,E2 -7159.045} C_VEL
LIN {X 0,Y 474.568,Z 246.871,A -85,B 0,C 180,E1 -7161.709,E2 -7161.709} C_VEL
LIN {X 0,Y 474.591,Z 246.865,A -85,B 0,C 180,E1 -7164.731,E2 -7164.731} C_VEL
LIN {X 0,Y 474.599,Z 246.864,A -85,B 0,C 180,E1 -7167.793,E2 -7167.793} C_VEL
LIN {X 0,Y 474.591,Z 246.868,A -85,B 0,C 180,E1 -7170.89,E2 -7170.89} C_VEL
LIN {X 0,Y 474.625,Z 246.861,A -85,B 0,C 180,E1 -7173.634,E2 -7173.634} C_VEL
LIN {X 0,Y 474.607,Z 246.865,A -85,B 0,C 180,E1 -7176.647,E2 -7176.647} C_VEL
LIN {X 0,Y 474.627,Z 246.859,A -85,B 0,C 180,E1 -7180.095,E2 -7180.095} C_VEL
LIN {X 0,Y 474.612,Z 246.868,A -85,B 0,C 180,E1 -7182.779,E2 -7182.779} C_VEL
LIN {X 0,Y 474.617,Z 246.861,A -85,B 0,C 180,E1 -7185.426,E2 -7185.426} C_VEL
LIN {X 0,Y 474.686,Z 246.853,A -85,B 0,C 180,E1 -7188.043,E2 -7188.043} C_VEL
LIN {X 0,Y 474.695,Z 246.85,A -85,B 0,C 180,E1 -7191.491,E2 -7191.491} C_VEL
LIN {X 0,Y 474.746,Z 246.847,A -85,B 0,C 180,E1 -7194.057,E2 -7194.057} C_VEL
LIN {X 0,Y 474.872,Z 246.828,A -85,B 0,C 180,E1 -7197.46,E2 -7197.46} C_VEL
LIN {X 0,Y 474.87,Z 246.833,A -85,B 0,C 180,E1 -7200.005,E2 -7200.005} C_VEL
LIN {X 0,Y 474.865,Z 246.833,A -85,B 0,C 180,E1 -7202.55,E2 -7202.55} C_VEL
LIN {X 0,Y 474.732,Z 246.851,A -85,B 0,C 180,E1 -7205.953,E2 -7205.953} C_VEL
LIN {X 0,Y 474.692,Z 246.853,A -85,B 0,C 180,E1 -7208.519,E2 -7208.519} C_VEL
LIN {X 0,Y 474.703,Z 246.858,A -85,B 0,C 180,E1 -7211.967,E2 -7211.967} C_VEL
LIN {X 0,Y 474.688,Z 246.854,A -85,B 0,C 180,E1 -7215.46,E2 -7215.46} C_VEL
LIN {X 0,Y 474.659,Z 246.855,A -85,B 0,C 180,E1 -7219.014,E2 -7219.014} C_VEL
LIN {X 0,Y 474.589,Z 246.871,A -85,B 0,C 180,E1 -7221.733,E2 -7221.733} C_VEL
LIN {X 0,Y 474.629,Z 246.859,A -85,B 0,C 180,E1 -7224.498,E2 -7224.498} C_VEL
LIN {X 0,Y 474.603,Z 246.868,A -85,B 0,C 180,E1 -7227.33,E2 -7227.33} C_VEL
LIN {X 0,Y 474.6,Z 246.863,A -85,B 0,C 180,E1 -7230.234,E2 -7230.234} C_VEL
LIN {X 0,Y 474.621,Z 246.867,A -85,B 0,C 180,E1 -7233.225,E2 -7233.225} C_VEL
LIN {X 0,Y 474.588,Z 246.867,A -85,B 0,C 180,E1 -7236.327,E2 -7236.327} C_VEL
LIN {X 0,Y 474.608,Z 246.868,A -85,B 0,C 180,E1 -7239.646,E2 -7239.646} C_VEL
LIN {X 0,Y 474.583,Z 246.871,A -85,B 0,C 180,E1 -7242.232,E2 -7242.232} C_VEL
LIN {X 0,Y 474.605,Z 247.169,A -85,B 0,C 180,E1 -7242.939,E2 -7242.939} C_VEL
LIN {X 0,Y 475.193,Z 250.81,A -85,B 0,C 180,E1 -7245.964,E2 -7245.964} C_VEL
LIN {X 0,Y 475.482,Z 253.899,A -85,B 0,C 180,E1 -7248.308,E2 -7248.308} C_VEL
LIN {X 0,Y 475.43,Z 257.06,A -85,B 0,C 180,E1 -7250.533,E2 -7250.533} C_VEL
LIN {X 0,Y 475.189,Z 260.813,A -85,B 0,C 180,E1 -7253.005,E2 -7253.005} C_VEL
LIN {X 0,Y 474.937,Z 265.557,A -85,B 0,C 180,E1 -7255.966,E2 -7255.966} C_VEL
LIN {X 0,Y 474.687,Z 270.355,A -85,B 0,C 180,E1 -7258.789,E2 -7258.789} C_VEL
LIN {X 0,Y 474.491,Z 275.547,A -85,B 0,C 180,E1 -7261.708,E2 -7261.708} C_VEL
LIN {X 0,Y 474.343,Z 281.041,A -85,B 0,C 180,E1 -7264.665,E2 -7264.665} C_VEL
LIN {X 0,Y 474.164,Z 286.165,A -85,B 0,C 180,E1 -7267.334,E2 -7267.334} C_VEL
LIN {X 0,Y 474.051,Z 291.668,A -85,B 0,C 180,E1 -7270.064,E2 -7270.064} C_VEL
LIN {X 0,Y 473.913,Z 297.155,A -85,B 0,C 180,E1 -7272.747,E2 -7272.747} C_VEL
LIN {X 0,Y 473.949,Z 301.557,A -85,B 0,C 180,E1 -7274.86,E2 -7274.86} C_VEL
LIN {X 0,Y 475.823,Z 311.677,A -85,B 0,C 180,E1 -7275.177,E2 -7275.177} C_VEL
LIN {X 0,Y 476.996,Z 319.721,A -85,B 0,C 180,E1 -7275.495,E2 -7275.495} C_VEL
LIN {X 0,Y 476.651,Z 330.349,A -85,B 0,C 180,E1 -7275.974,E2 -7275.974} C_VEL
LIN {X 0,Y 476.215,Z 340.474,A -85,B 0,C 180,E1 -7276.56,E2 -7276.56} C_VEL
LIN {X 0,Y 475.817,Z 349.446,A -85,B 0,C 180,E1 -7277.2,E2 -7277.2} C_VEL
LIN {X 0,Y 475.557,Z 358.235,A -85,B 0,C 180,E1 -7277.959,E2 -7277.959} C_VEL
LIN {X 0,Y 475.217,Z 365.521,A -85,B 0,C 180,E1 -7278.7,E2 -7278.7} C_VEL
LIN {X 0,Y 474.884,Z 372.713,A -85,B 0,C 180,E1 -7279.555,E2 -7279.555} C_VEL
LIN {X 0,Y 474.606,Z 378.889,A -85,B 0,C 180,E1 -7280.411,E2 -7280.411} C_VEL
LIN {X 0,Y 474.319,Z 385.396,A -85,B 0,C 180,E1 -7281.479,E2 -7281.479} C_VEL
LIN {X 0,Y 474.102,Z 389.875,A -85,B 0,C 180,E1 -7282.333,E2 -7282.333} C_VEL
LIN {X 0,Y 473.963,Z 394.809,A -85,B 0,C 180,E1 -7283.47,E2 -7283.47} C_VEL
LIN {X 0,Y 473.847,Z 399.628,A -85,B 0,C 180,E1 -7284.895,E2 -7284.895} C_VEL
LIN {X 0,Y 473.755,Z 401.974,A -85,B 0,C 180,E1 -7285.746,E2 -7285.746} C_VEL
LIN {X 0,Y 473.803,Z 403.76,A -85,B 0,C 180,E1 -7286.599,E2 -7286.599} C_VEL
LIN {X 0,Y 473.698,Z 406.186,A -85,B 0,C 180,E1 -7288.3,E2 -7288.3} C_VEL
LIN {X 0,Y 473.691,Z 406.769,A -85,B 0,C 180,E1 -7289.15,E2 -7289.15} C_VEL
LIN {X 0,Y 473.691,Z 406.769,A -85,B 0,C 180,E1 -7290.85,E2 -7290.85} C_VEL
LIN {X 0,Y 473.698,Z 406.186,A -85,B 0,C 180,E1 -7291.7,E2 -7291.7} C_VEL
LIN {X 0,Y 473.803,Z 403.76,A -85,B 0,C 180,E1 -7293.401,E2 -7293.401} C_VEL
LIN {X 0,Y 473.778,Z 400.836,A -85,B 0,C 180,E1 -7294.68,E2 -7294.68} C_VEL
LIN {X 0,Y 473.91,Z 396.877,A -85,B 0,C 180,E1 -7295.958,E2 -7295.958} C_VEL
LIN {X 0,Y 474.035,Z 391.78,A -85,B 0,C 180,E1 -7297.24,E2 -7297.24} C_VEL
LIN {X 0,Y 474.266,Z 386.546,A -85,B 0,C 180,E1 -7298.307,E2 -7298.307} C_VEL
LIN {X 0,Y 474.521,Z 380.259,A -85,B 0,C 180,E1 -7299.376,E2 -7299.376} C_VEL
LIN {X 0,Y 474.796,Z 374.334,A -85,B 0,C 180,E1 -7300.231,E2 -7300.231} C_VEL
LIN {X 0,Y 475.086,Z 367.433,A -85,B 0,C 180,E1 -7301.087,E2 -7301.087} C_VEL
LIN {X 0,Y 475.502,Z 359.281,A -85,B 0,C 180,E1 -7301.942,E2 -7301.942} C_VEL
LIN {X 0,Y 475.815,Z 350.866,A -85,B 0,C 180,E1 -7302.686,E2 -7302.686} C_VEL
LIN {X 0,Y 476.157,Z 342.588,A -85,B 0,C 180,E1 -7303.301,E2 -7303.301} C_VEL
LIN {X 0,Y 476.545,Z 332.359,A -85,B 0,C 180,E1 -7303.92,E2 -7303.92} C_VEL
LIN {X 0,Y 476.874,Z 323.58,A -85,B 0,C 180,E1 -7304.346,E2 -7304.346} C_VEL
LIN {X 0,Y 476.849,Z 318.458,A -85,B 0,C 180,E1 -7304.564,E2 -7304.564} C_VEL
LIN {X 0,Y 474.545,Z 305.016,A -85,B 0,C 180,E1 -7305.05,E2 -7305.05} C_VEL
LIN {X 0,Y 473.928,Z 301.455,A -85,B 0,C 180,E1 -7305.168,E2 -7305.168} C_VEL
LIN {X 0,Y 474.004,Z 294.826,A -85,B 0,C 180,E1 -7308.387,E2 -7308.387} C_VEL
LIN {X 0,Y 474.151,Z 289.591,A -85,B 0,C 180,E1 -7310.96,E2 -7310.96} C_VEL
LIN {X 0,Y 474.201,Z 284.358,A -85,B 0,C 180,E1 -7313.588,E2 -7313.588} C_VEL
LIN {X 0,Y 474.4,Z 279.051,A -85,B 0,C 180,E1 -7316.387,E2 -7316.387} C_VEL
LIN {X 0,Y 474.544,Z 273.782,A -85,B 0,C 180,E1 -7319.257,E2 -7319.257} C_VEL
LIN {X 0,Y 474.815,Z 268.178,A -85,B 0,C 180,E1 -7322.465,E2 -7322.465} C_VEL
LIN {X 0,Y 475.067,Z 263.073,A -85,B 0,C 180,E1 -7325.542,E2 -7325.542} C_VEL
LIN {X 0,Y 475.382,Z 258.616,A -85,B 0,C 180,E1 -7328.41,E2 -7328.41} C_VEL
LIN {X 0,Y 475.514,Z 254.726,A -85,B 0,C 180,E1 -7331.079,E2 -7331.079} C_VEL
LIN {X 0,Y 475.285,Z 251.406,A -85,B 0,C 180,E1 -7333.564,E2 -7333.564} C_VEL
LIN {X 0,Y 474.718,Z 247.834,A -85,B 0,C 180,E1 -7336.503,E2 -7336.503} C_VEL
LIN {X 0,Y 474.604,Z 247.182,A -85,B 0,C 180,E1 -7337.061,E2 -7337.061} C_VEL
LIN {X 0,Y 474.599,Z 246.869,A -85,B 0,C 180,E1 -7338.209,E2 -7338.209} C_VEL
LIN {X 0,Y 474.625,Z 246.865,A -85,B 0,C 180,E1 -7340.449,E2 -7340.449} C_VEL
LIN {X 0,Y 474.588,Z 246.864,A -85,B 0,C 180,E1 -7343.673,E2 -7343.673} C_VEL
LIN {X 0,Y 474.621,Z 246.867,A -85,B 0,C 180,E1 -7346.775,E2 -7346.775} C_VEL
LIN {X 0,Y 474.6,Z 246.863,A -85,B 0,C 180,E1 -7349.766,E2 -7349.766} C_VEL
LIN {X 0,Y 474.607,Z 246.867,A -85,B 0,C 180,E1 -7352.681,E2 -7352.681} C_VEL
LIN {X 0,Y 474.629,Z 246.859,A -85,B 0,C 180,E1 -7355.502,E2 -7355.502} C_VEL
LIN {X 0,Y 474.627,Z 246.86,A -85,B 0,C 180,E1 -7358.883,E2 -7358.883} C_VEL
LIN {X 0,Y 474.631,Z 246.862,A -85,B 0,C 180,E1 -7361.879,E2 -7361.879} C_VEL
LIN {X 0,Y 474.688,Z 246.854,A -85,B 0,C 180,E1 -7364.54,E2 -7364.54} C_VEL
LIN {X 0,Y 474.703,Z 246.858,A -85,B 0,C 180,E1 -7368.033,E2 -7368.033} C_VEL
LIN {X 0,Y 474.692,Z 246.853,A -85,B 0,C 180,E1 -7371.481,E2 -7371.481} C_VEL
LIN {X 0,Y 474.732,Z 246.851,A -85,B 0,C 180,E1 -7374.047,E2 -7374.047} C_VEL
LIN {X 0,Y 474.865,Z 246.833,A -85,B 0,C 180,E1 -7377.45,E2 -7377.45} C_VEL
LIN {X 0,Y 474.87,Z 246.833,A -85,B 0,C 180,E1 -7379.995,E2 -7379.995} C_VEL
LIN {X 0,Y 474.872,Z 246.828,A -85,B 0,C 180,E1 -7382.54,E2 -7382.54} C_VEL
LIN {X 0,Y 474.746,Z 246.847,A -85,B 0,C 180,E1 -7385.943,E2 -7385.943} C_VEL
LIN {X 0,Y 474.695,Z 246.85,A -85,B 0,C 180,E1 -7388.509,E2 -7388.509} C_VEL
LIN {X 0,Y 474.686,Z 246.853,A -85,B 0,C 180,E1 -7391.957,E2 -7391.957} C_VEL
LIN {X 0,Y 474.659,Z 246.857,A -85,B 0,C 180,E1 -7395.762,E2 -7395.762} C_VEL
LIN {X 0,Y 474.637,Z 246.864,A -85,B 0,C 180,E1 -7399.005,E2 -7399.005} C_VEL
LIN {X 0,Y 474.561,Z 246.868,A -85,B 0,C 180,E1 -7401.724,E2 -7401.724} C_VEL
LIN {X 0,Y 474.62,Z 246.862,A -85,B 0,C 180,E1 -7404.488,E2 -7404.488} C_VEL
LIN {X 0,Y 474.65,Z 246.858,A -85,B 0,C 180,E1 -7407.329,E2 -7407.329} C_VEL
LIN {X 0,Y 474.57,Z 246.868,A -85,B 0,C 180,E1 -7410.225,E2 -7410.225} C_VEL
LIN {X 0,Y 474.606,Z 246.863,A -85,B 0,C 180,E1 -7413.215,E2 -7413.215} C_VEL
LIN {X 0,Y 474.553,Z 246.872,A -85,B 0,C 180,E1 -7416.318,E2 -7416.318} C_VEL
LIN {X 0,Y 474.574,Z 246.866,A -85,B 0,C 180,E1 -7419.641,E2 -7419.641} C_VEL
LIN {X 0,Y 474.606,Z 246.863,A -85,B 0,C 180,E1 -7422.925,E2 -7422.925} C_VEL
LIN {X 0,Y 474.57,Z 246.869,A -85,B 0,C 180,E1 -7425.891,E2 -7425.891} C_VEL
LIN {X 0,Y 474.594,Z 246.863,A -85,B 0,C 180,E1 -7429.034,E2 -7429.034} C_VEL
LIN {X 0,Y 474.566,Z 246.869,A -85,B 0,C 180,E1 -7431.698,E2 -7431.698} C_VEL
LIN {X 0,Y 474.574,Z 246.866,A -85,B 0,C 180,E1 -7434.722,E2 -7434.722} C_VEL
LIN {X 0,Y 474.583,Z 246.87,A -85,B 0,C 180,E1 -7437.784,E2 -7437.784} C_VEL
LIN {X 0,Y 474.573,Z 246.866,A -85,B 0,C 180,E1 -7440.879,E2 -7440.879} C_VEL
LIN {X 0,Y 474.608,Z 246.867,A -85,B 0,C 180,E1 -7443.626,E2 -7443.626} C_VEL
LIN {X 0,Y 474.592,Z 246.863,A -85,B 0,C 180,E1 -7446.633,E2 -7446.633} C_VEL
LIN {X 0,Y 474.612,Z 246.863,A -85,B 0,C 180,E1 -7449.183,E2 -7449.183} C_VEL
LIN {X 0,Y 474.602,Z 246.867,A -85,B 0,C 180,E1 -7451.632,E2 -7451.632} C_VEL
LIN {X 0,Y 473.944,Z 246.951,A -85,B 0,C 180,E1 -7452.341,E2 -7452.341} C_VEL
LIN {X 0,Y 471.099,Z 247.309,A -85,B 0,C 180,E1 -7453.493,E2 -7453.493} C_VEL
LIN {X 0,Y 468.684,Z 247.609,A -85,B 0,C 180,E1 -7454.421,E2 -7454.421} C_VEL
LIN {X 0,Y 467.64,Z 247.736,A -85,B 0,C 180,E1 -7455.138,E2 -7455.138} C_VEL
LIN {X 0,Y 467.552,Z 247.745,A -85,B 0,C 180,E1 -7455.381,E2 -7455.381} C_VEL
LIN {X 0,Y 467.631,Z 247.734,A -85,B 0,C 180,E1 -7457.854,E2 -7457.854} C_VEL
LIN {X 0,Y 467.631,Z 247.738,A -85,B 0,C 180,E1 -7461.356,E2 -7461.356} C_VEL
LIN {X 0,Y 467.696,Z 247.726,A -85,B 0,C 180,E1 -7463.962,E2 -7463.962} C_VEL
LIN {X 0,Y 467.801,Z 247.716,A -85,B 0,C 180,E1 -7467.417,E2 -7467.417} C_VEL
LIN {X 0,Y 467.813,Z 247.712,A -85,B 0,C 180,E1 -7470,E2 -7470} C_VEL
LIN {X 0,Y 467.801,Z 247.716,A -85,B 0,C 180,E1 -7472.583,E2 -7472.583} C_VEL
LIN {X 0,Y 467.696,Z 247.726,A -85,B 0,C 180,E1 -7476.038,E2 -7476.038} C_VEL
LIN {X 0,Y 467.631,Z 247.738,A -85,B 0,C 180,E1 -7478.644,E2 -7478.644} C_VEL
LIN {X 0,Y 467.625,Z 247.737,A -85,B 0,C 180,E1 -7482.38,E2 -7482.38} C_VEL
LIN {X 0,Y 467.612,Z 247.737,A -85,B 0,C 180,E1 -7485.899,E2 -7485.899} C_VEL
LIN {X 0,Y 467.562,Z 247.739,A -85,B 0,C 180,E1 -7489.31,E2 -7489.31} C_VEL
LIN {X 0,Y 467.515,Z 247.749,A -85,B 0,C 180,E1 -7492.074,E2 -7492.074} C_VEL
LIN {X 0,Y 467.56,Z 247.74,A -85,B 0,C 180,E1 -7494.889,E2 -7494.889} C_VEL
LIN {X 0,Y 467.568,Z 247.741,A -85,B 0,C 180,E1 -7497.772,E2 -7497.772} C_VEL
LIN {X 0,Y 467.518,Z 247.744,A -85,B 0,C 180,E1 -7501.05,E2 -7501.05} C_VEL
LIN {X 0,Y 467.534,Z 247.747,A -85,B 0,C 180,E1 -7504.246,E2 -7504.246} C_VEL
LIN {X 0,Y 467.497,Z 247.748,A -85,B 0,C 180,E1 -7507.191,E2 -7507.191} C_VEL
LIN {X 0,Y 467.546,Z 247.743,A -85,B 0,C 180,E1 -7510.267,E2 -7510.267} C_VEL
LIN {X 0,Y 467.57,Z 247.738,A -85,B 0,C 180,E1 -7512.576,E2 -7512.576} C_VEL
LIN {X 0,Y 467.53,Z 247.744,A -85,B 0,C 180,E1 -7516.263,E2 -7516.263} C_VEL
LIN {X 0,Y 467.54,Z 247.742,A -85,B 0,C 180,E1 -7518.727,E2 -7518.727} C_VEL
LIN {X 0,Y 467.524,Z 247.746,A -85,B 0,C 180,E1 -7521.961,E2 -7521.961} C_VEL
LIN {X 0,Y 467.53,Z 247.749,A -85,B 0,C 180,E1 -7525.173,E2 -7525.173} C_VEL
LIN {X 0,Y 467.546,Z 247.741,A -85,B 0,C 180,E1 -7528.265,E2 -7528.265} C_VEL
LIN {X 0,Y 467.544,Z 247.748,A -85,B 0,C 180,E1 -7531.256,E2 -7531.256} C_VEL
LIN {X 0,Y 467.569,Z 247.738,A -85,B 0,C 180,E1 -7534.165,E2 -7534.165} C_VEL
LIN {X 0,Y 467.548,Z 247.749,A -85,B 0,C 180,E1 -7537.001,E2 -7537.001} C_VEL
LIN {X 0,Y 467.596,Z 247.735,A -85,B 0,C 180,E1 -7539.783,E2 -7539.783} C_VEL
LIN {X 0,Y 467.572,Z 247.741,A -85,B 0,C 180,E1 -7542.512,E2 -7542.512} C_VEL
LIN {X 0,Y 467.577,Z 247.74,A -85,B 0,C 180,E1 -7545.202,E2 -7545.202} C_VEL
LIN {X 0,Y 467.638,Z 247.73,A -85,B 0,C 180,E1 -7547.86,E2 -7547.86} C_VEL
LIN {X 0,Y 467.653,Z 247.728,A -85,B 0,C 180,E1 -7551.362,E2 -7551.362} C_VEL
LIN {X 0,Y 467.711,Z 247.722,A -85,B 0,C 180,E1 -7553.968,E2 -7553.968} C_VEL
LIN {X 0,Y 467.837,Z 247.705,A -85,B 0,C 180,E1 -7557.422,E2 -7557.422} C_VEL
LIN {X 0,Y 467.839,Z 247.708,A -85,B 0,C 180,E1 -7560.005,E2 -7560.005} C_VEL
LIN {X 0,Y 467.805,Z 247.712,A -85,B 0,C 180,E1 -7562.588,E2 -7562.588} C_VEL
LIN {X 0,Y 467.697,Z 247.729,A -85,B 0,C 180,E1 -7566.043,E2 -7566.043} C_VEL
LIN {X 0,Y 467.653,Z 247.729,A -85,B 0,C 180,E1 -7568.648,E2 -7568.648} C_VEL
LIN {X 0,Y 467.655,Z 247.733,A -85,B 0,C 180,E1 -7572.15,E2 -7572.15} C_VEL
LIN {X 0,Y 467.613,Z 247.739,A -85,B 0,C 180,E1 -7575.7,E2 -7575.7} C_VEL
LIN {X 0,Y 467.618,Z 247.735,A -85,B 0,C 180,E1 -7579.312,E2 -7579.312} C_VEL
LIN {X 0,Y 467.533,Z 247.745,A -85,B 0,C 180,E1 -7582.078,E2 -7582.078} C_VEL
LIN {X 0,Y 467.563,Z 247.74,A -85,B 0,C 180,E1 -7584.894,E2 -7584.894} C_VEL
LIN {X 0,Y 467.549,Z 247.745,A -85,B 0,C 180,E1 -7587.777,E2 -7587.777} C_VEL
LIN {X 0,Y 467.553,Z 247.744,A -85,B 0,C 180,E1 -7591.043,E2 -7591.043} C_VEL
LIN {X 0,Y 467.582,Z 247.739,A -85,B 0,C 180,E1 -7594.243,E2 -7594.243} C_VEL
LIN {X 0,Y 467.544,Z 247.749,A -85,B 0,C 180,E1 -7597.187,E2 -7597.187} C_VEL
LIN {X 0,Y 467.564,Z 247.745,A -85,B 0,C 180,E1 -7600.27,E2 -7600.27} C_VEL
LIN {X 0,Y 467.57,Z 247.996,A -85,B 0,C 180,E1 -7602.566,E2 -7602.566} C_VEL
LIN {X 0,Y 468.044,Z 250.958,A -85,B 0,C 180,E1 -7605.112,E2 -7605.112} C_VEL
LIN {X 0,Y 468.427,Z 254.006,A -85,B 0,C 180,E1 -7607.535,E2 -7607.535} C_VEL
LIN {X 0,Y 468.465,Z 257.297,A -85,B 0,C 180,E1 -7609.921,E2 -7609.921} C_VEL
LIN {X 0,Y 468.278,Z 260.353,A -85,B 0,C 180,E1 -7612.025,E2 -7612.025} C_VEL
LIN {X 0,Y 467.951,Z 265.297,A -85,B 0,C 180,E1 -7615.201,E2 -7615.201} C_VEL
LIN {X 0,Y 467.699,Z 270.343,A -85,B 0,C 180,E1 -7618.269,E2 -7618.269} C_VEL
LIN {X 0,Y 467.45,Z 275.514,A -85,B 0,C 180,E1 -7621.243,E2 -7621.243} C_VEL
LIN {X 0,Y 467.308,Z 280.769,A -85,B 0,C 180,E1 -7624.143,E2 -7624.143} C_VEL
LIN {X 0,Y 467.124,Z 286.095,A -85,B 0,C 180,E1 -7626.973,E2 -7626.973} C_VEL
LIN {X 0,Y 467.01,Z 291.563,A -85,B 0,C 180,E1 -7629.75,E2 -7629.75} C_VEL
LIN {X 0,Y 466.862,Z 297.043,A -85,B 0,C 180,E1 -7632.478,E2 -7632.478} C_VEL
LIN {X 0,Y 466.837,Z 301.487,A -85,B 0,C 180,E1 -7634.626,E2 -7634.626} C_VEL
LIN {X 0,Y 468.781,Z 311.906,A -85,B 0,C 180,E1 -7634.963,E2 -7634.963} C_VEL
LIN {X 0,Y 470.077,Z 320.852,A -85,B 0,C 180,E1 -7635.332,E2 -7635.332} C_VEL
LIN {X 0,Y 469.724,Z 331.219,A -85,B 0,C 180,E1 -7635.818,E2 -7635.818} C_VEL
LIN {X 0,Y 469.304,Z 340.358,A -85,B 0,C 180,E1 -7636.358,E2 -7636.358} C_VEL
LIN {X 0,Y 468.877,Z 349.355,A -85,B 0,C 180,E1 -7637.007,E2 -7637.007} C_VEL
LIN {X 0,Y 468.646,Z 357.276,A -85,B 0,C 180,E1 -7637.692,E2 -7637.692} C_VEL
LIN {X 0,Y 468.252,Z 365.491,A -85,B 0,C 180,E1 -7638.529,E2 -7638.529} C_VEL
LIN {X 0,Y 467.883,Z 372.708,A -85,B 0,C 180,E1 -7639.397,E2 -7639.397} C_VEL
LIN {X 0,Y 467.583,Z 378.885,A -85,B 0,C 180,E1 -7640.265,E2 -7640.265} C_VEL
LIN {X 0,Y 467.291,Z 385.392,A -85,B 0,C 180,E1 -7641.35,E2 -7641.35} C_VEL
LIN {X 0,Y 467.048,Z 389.87,A -85,B 0,C 180,E1 -7642.217,E2 -7642.217} C_VEL
LIN {X 0,Y 466.871,Z 395.23,A -85,B 0,C 180,E1 -7643.49,E2 -7643.49} C_VEL
LIN {X 0,Y 466.785,Z 399.624,A -85,B 0,C 180,E1 -7644.817,E2 -7644.817} C_VEL
LIN {X 0,Y 466.666,Z 401.972,A -85,B 0,C 180,E1 -7645.682,E2 -7645.682} C_VEL
LIN {X 0,Y 466.698,Z 403.757,A -85,B 0,C 180,E1 -7646.547,E2 -7646.547} C_VEL
LIN {X 0,Y 466.608,Z 406.182,A -85,B 0,C 180,E1 -7648.274,E2 -7648.274} C_VEL
LIN {X 0,Y 466.593,Z 406.765,A -85,B 0,C 180,E1 -7649.137,E2 -7649.137} C_VEL
LIN {X 0,Y 466.593,Z 406.765,A -85,B 0,C 180,E1 -7650.863,E2 -7650.863} C_VEL
LIN {X 0,Y 466.608,Z 406.182,A -85,B 0,C 180,E1 -7651.726,E2 -7651.726} C_VEL
LIN {X 0,Y 466.698,Z 403.757,A -85,B 0,C 180,E1 -7653.453,E2 -7653.453} C_VEL
LIN {X 0,Y 466.705,Z 400.832,A -85,B 0,C 180,E1 -7654.751,E2 -7654.751} C_VEL
LIN {X 0,Y 466.815,Z 396.873,A -85,B 0,C 180,E1 -7656.049,E2 -7656.049} C_VEL
LIN {X 0,Y 466.965,Z 391.775,A -85,B 0,C 180,E1 -7657.35,E2 -7657.35} C_VEL
LIN {X 0,Y 467.209,Z 386.542,A -85,B 0,C 180,E1 -7658.434,E2 -7658.434} C_VEL
LIN {X 0,Y 467.49,Z 380.255,A -85,B 0,C 180,E1 -7659.518,E2 -7659.518} C_VEL
LIN {X 0,Y 467.778,Z 374.329,A -85,B 0,C 180,E1 -7660.386,E2 -7660.386} C_VEL
LIN {X 0,Y 468.115,Z 367.41,A -85,B 0,C 180,E1 -7661.255,E2 -7661.255} C_VEL
LIN {X 0,Y 468.55,Z 359.227,A -85,B 0,C 180,E1 -7662.122,E2 -7662.122} C_VEL
LIN {X 0,Y 468.844,Z 350.78,A -85,B 0,C 180,E1 -7662.878,E2 -7662.878} C_VEL
LIN {X 0,Y 469.247,Z 341.993,A -85,B 0,C 180,E1 -7663.533,E2 -7663.533} C_VEL
LIN {X 0,Y 469.666,Z 332.225,A -85,B 0,C 180,E1 -7664.128,E2 -7664.128} C_VEL
LIN {X 0,Y 470.037,Z 322.141,A -85,B 0,C 180,E1 -7664.614,E2 -7664.614} C_VEL
LIN {X 0,Y 469.26,Z 314.77,A -85,B 0,C 180,E1 -7664.931,E2 -7664.931} C_VEL
LIN {X 0,Y 467.137,Z 303.242,A -85,B 0,C 180,E1 -7665.327,E2 -7665.327} C_VEL
LIN {X 0,Y 466.841,Z 301.315,A -85,B 0,C 180,E1 -7665.403,E2 -7665.403} C_VEL
LIN {X 0,Y 466.926,Z 295.059,A -85,B 0,C 180,E1 -7668.508,E2 -7668.508} C_VEL
LIN {X 0,Y 467.085,Z 289.73,A -85,B 0,C 180,E1 -7671.168,E2 -7671.168} C_VEL
LIN {X 0,Y 467.156,Z 284.306,A -85,B 0,C 180,E1 -7673.965,E2 -7673.965} C_VEL
LIN {X 0,Y 467.354,Z 278.99,A -85,B 0,C 180,E1 -7676.816,E2 -7676.816} C_VEL
LIN {X 0,Y 467.529,Z 273.759,A -85,B 0,C 180,E1 -7679.739,E2 -7679.739} C_VEL
LIN {X 0,Y 467.79,Z 268.635,A -85,B 0,C 180,E1 -7682.741,E2 -7682.741} C_VEL
LIN {X 0,Y 468.051,Z 263.61,A -85,B 0,C 180,E1 -7685.845,E2 -7685.845} C_VEL
LIN {X 0,Y 468.397,Z 258.728,A -85,B 0,C 180,E1 -7689.063,E2 -7689.063} C_VEL
LIN {X 0,Y 468.51,Z 255.423,A -85,B 0,C 180,E1 -7691.403,E2 -7691.403} C_VEL
LIN {X 0,Y 468.246,Z 252.168,A -85,B 0,C 180,E1 -7693.906,E2 -7693.906} C_VEL
LIN {X 0,Y 467.768,Z 249.323,A -85,B 0,C 180,E1 -7696.277,E2 -7696.277} C_VEL
LIN {X 0,Y 467.57,Z 247.997,A -85,B 0,C 180,E1 -7697.434,E2 -7697.434} C_VEL
LIN {X 0,Y 467.569,Z 247.744,A -85,B 0,C 180,E1 -7700.046,E2 -7700.046} C_VEL
LIN {X 0,Y 467.527,Z 247.749,A -85,B 0,C 180,E1 -7703.034,E2 -7703.034} C_VEL
LIN {X 0,Y 467.573,Z 247.74,A -85,B 0,C 180,E1 -7706.207,E2 -7706.207} C_VEL
LIN {X 0,Y 467.569,Z 247.739,A -85,B 0,C 180,E1 -7709.262,E2 -7709.262} C_VEL
LIN {X 0,Y 467.554,Z 247.748,A -85,B 0,C 180,E1 -7712.478,E2 -7712.478} C_VEL
LIN {X 0,Y 467.563,Z 247.74,A -85,B 0,C 180,E1 -7715.106,E2 -7715.106} C_VEL
LIN {X 0,Y 467.533,Z 247.745,A -85,B 0,C 180,E1 -7717.922,E2 -7717.922} C_VEL
LIN {X 0,Y 467.618,Z 247.735,A -85,B 0,C 180,E1 -7720.688,E2 -7720.688} C_VEL
LIN {X 0,Y 467.613,Z 247.739,A -85,B 0,C 180,E1 -7724.3,E2 -7724.3} C_VEL
LIN {X 0,Y 467.655,Z 247.733,A -85,B 0,C 180,E1 -7727.85,E2 -7727.85} C_VEL
LIN {X 0,Y 467.653,Z 247.729,A -85,B 0,C 180,E1 -7731.352,E2 -7731.352} C_VEL
LIN {X 0,Y 467.697,Z 247.729,A -85,B 0,C 180,E1 -7733.957,E2 -7733.957} C_VEL
LIN {X 0,Y 467.805,Z 247.712,A -85,B 0,C 180,E1 -7737.412,E2 -7737.412} C_VEL
LIN {X 0,Y 467.839,Z 247.708,A -85,B 0,C 180,E1 -7739.995,E2 -7739.995} C_VEL
LIN {X 0,Y 467.837,Z 247.705,A -85,B 0,C 180,E1 -7742.578,E2 -7742.578} C_VEL
LIN {X 0,Y 467.711,Z 247.722,A -85,B 0,C 180,E1 -7746.032,E2 -7746.032} C_VEL
LIN {X 0,Y 467.653,Z 247.728,A -85,B 0,C 180,E1 -7748.638,E2 -7748.638} C_VEL
LIN {X 0,Y 467.638,Z 247.73,A -85,B 0,C 180,E1 -7752.14,E2 -7752.14} C_VEL
LIN {X 0,Y 467.628,Z 247.732,A -85,B 0,C 180,E1 -7755.879,E2 -7755.879} C_VEL
LIN {X 0,Y 467.597,Z 247.74,A -85,B 0,C 180,E1 -7759.302,E2 -7759.302} C_VEL
LIN {X 0,Y 467.507,Z 247.746,A -85,B 0,C 180,E1 -7762.068,E2 -7762.068} C_VEL
LIN {X 0,Y 467.562,Z 247.746,A -85,B 0,C 180,E1 -7764.883,E2 -7764.883} C_VEL
LIN {X 0,Y 467.588,Z 247.736,A -85,B 0,C 180,E1 -7767.764,E2 -7767.764} C_VEL
LIN {X 0,Y 467.533,Z 247.747,A -85,B 0,C 180,E1 -7771.039,E2 -7771.039} C_VEL
LIN {X 0,Y 467.552,Z 247.743,A -85,B 0,C 180,E1 -7774.237,E2 -7774.237} C_VEL
LIN {X 0,Y 467.509,Z 247.747,A -85,B 0,C 180,E1 -7777.181,E2 -7777.181} C_VEL
LIN {X 0,Y 467.532,Z 247.748,A -85,B 0,C 180,E1 -7780.26,E2 -7780.26} C_VEL
LIN {X 0,Y 467.574,Z 247.743,A -85,B 0,C 180,E1 -7782.566,E2 -7782.566} C_VEL
LIN {X 0,Y 467.528,Z 247.751,A -85,B 0,C 180,E1 -7786.253,E2 -7786.253} C_VEL
LIN {X 0,Y 467.539,Z 247.744,A -85,B 0,C 180,E1 -7788.717,E2 -7788.717} C_VEL
LIN {X 0,Y 467.525,Z 247.744,A -85,B 0,C 180,E1 -7791.402,E2 -7791.402} C_VEL
LIN {X 0,Y 467.508,Z 247.751,A -85,B 0,C 180,E1 -7794.256,E2 -7794.256} C_VEL
LIN {X 0,Y 467.526,Z 247.744,A -85,B 0,C 180,E1 -7797.317,E2 -7797.317} C_VEL
LIN {X 0,Y 467.52,Z 247.745,A -85,B 0,C 180,E1 -7800.662,E2 -7800.662} C_VEL
LIN {X 0,Y 467.568,Z 247.739,A -85,B 0,C 180,E1 -7803.197,E2 -7803.197} C_VEL
LIN {X 0,Y 467.532,Z 247.746,A -85,B 0,C 180,E1 -7806.055,E2 -7806.055} C_VEL
LIN {X 0,Y 467.578,Z 247.737,A -85,B 0,C 180,E1 -7808.855,E2 -7808.855} C_VEL
LIN {X 0,Y 467.576,Z 247.745,A -85,B 0,C 180,E1 -7811.623,E2 -7811.623} C_VEL
LIN {X 0,Y 467.603,Z 247.737,A -85,B 0,C 180,E1 -7814.304,E2 -7814.304} C_VEL
LIN {X 0,Y 467.552,Z 247.745,A -85,B 0,C 180,E1 -7815.381,E2 -7815.381} C_VEL
LIN {X 0,Y 466.88,Z 247.829,A -85,B 0,C 180,E1 -7816.101,E2 -7816.101} C_VEL
LIN {X 0,Y 464.042,Z 248.185,A -85,B 0,C 180,E1 -7817.27,E2 -7817.27} C_VEL
LIN {X 0,Y 461.646,Z 248.48,A -85,B 0,C 180,E1 -7818.212,E2 -7818.212} C_VEL
LIN {X 0,Y 460.615,Z 248.61,A -85,B 0,C 180,E1 -7818.94,E2 -7818.94} C_VEL
LIN {X 0,Y 460.53,Z 248.619,A -85,B 0,C 180,E1 -7819.187,E2 -7819.187} C_VEL
LIN {X 0,Y 460.663,Z 248.603,A -85,B 0,C 180,E1 -7822.528,E2 -7822.528} C_VEL
LIN {X 0,Y 460.643,Z 248.606,A -85,B 0,C 180,E1 -7824.748,E2 -7824.748} C_VEL
LIN {X 0,Y 460.766,Z 248.592,A -85,B 0,C 180,E1 -7827.377,E2 -7827.377} C_VEL
LIN {X 0,Y 460.784,Z 248.588,A -85,B 0,C 180,E1 -7830,E2 -7830} C_VEL
LIN {X 0,Y 460.766,Z 248.592,A -85,B 0,C 180,E1 -7832.623,E2 -7832.623} C_VEL
LIN {X 0,Y 460.662,Z 248.603,A -85,B 0,C 180,E1 -7836.13,E2 -7836.13} C_VEL
LIN {X 0,Y 460.598,Z 248.614,A -85,B 0,C 180,E1 -7838.777,E2 -7838.777} C_VEL
LIN {X 0,Y 460.568,Z 248.616,A -85,B 0,C 180,E1 -7842.458,E2 -7842.458} C_VEL
LIN {X 0,Y 460.557,Z 248.617,A -85,B 0,C 180,E1 -7846.009,E2 -7846.009} C_VEL
LIN {X 0,Y 460.512,Z 248.622,A -85,B 0,C 180,E1 -7848.906,E2 -7848.906} C_VEL
LIN {X 0,Y 460.502,Z 248.619,A -85,B 0,C 180,E1 -7851.486,E2 -7851.486} C_VEL
LIN {X 0,Y 460.498,Z 248.626,A -85,B 0,C 180,E1 -7854.334,E2 -7854.334} C_VEL
LIN {X 0,Y 460.524,Z 248.616,A -85,B 0,C 180,E1 -7857.246,E2 -7857.246} C_VEL
LIN {X 0,Y 460.471,Z 248.628,A -85,B 0,C 180,E1 -7860.242,E2 -7860.242} C_VEL
LIN {X 0,Y 460.473,Z 248.623,A -85,B 0,C 180,E1 -7863.329,E2 -7863.329} C_VEL
LIN {X 0,Y 460.425,Z 248.629,A -85,B 0,C 180,E1 -7866.533,E2 -7866.533} C_VEL
LIN {X 0,Y 460.527,Z 248.623,A -85,B 0,C 180,E1 -7869.862,E2 -7869.862} C_VEL
LIN {X 0,Y 460.494,Z 248.62,A -85,B 0,C 180,E1 -7872.909,E2 -7872.909} C_VEL
LIN {X 0,Y 460.477,Z 248.627,A -85,B 0,C 180,E1 -7875.834,E2 -7875.834} C_VEL
LIN {X 0,Y 460.491,Z 248.622,A -85,B 0,C 180,E1 -7878.994,E2 -7878.994} C_VEL
LIN {X 0,Y 460.476,Z 248.627,A -85,B 0,C 180,E1 -7881.271,E2 -7881.271} C_VEL
LIN {X 0,Y 460.474,Z 248.622,A -85,B 0,C 180,E1 -7884.56,E2 -7884.56} C_VEL
LIN {X 0,Y 460.495,Z 248.622,A -85,B 0,C 180,E1 -7887.721,E2 -7887.721} C_VEL
LIN {X 0,Y 460.506,Z 248.621,A -85,B 0,C 180,E1 -7890.775,E2 -7890.775} C_VEL
LIN {X 0,Y 460.527,Z 248.616,A -85,B 0,C 180,E1 -7893.74,E2 -7893.74} C_VEL
LIN {X 0,Y 460.517,Z 248.62,A -85,B 0,C 180,E1 -7896.63,E2 -7896.63} C_VEL
LIN {X 0,Y 460.525,Z 248.617,A -85,B 0,C 180,E1 -7899.458,E2 -7899.458} C_VEL
LIN {X 0,Y 460.524,Z 248.617,A -85,B 0,C 180,E1 -7902.235,E2 -7902.235} C_VEL
LIN {X 0,Y 460.538,Z 248.619,A -85,B 0,C 180,E1 -7904.97,E2 -7904.97} C_VEL
LIN {X 0,Y 460.592,Z 248.614,A -85,B 0,C 180,E1 -7908.565,E2 -7908.565} C_VEL
LIN {X 0,Y 460.603,Z 248.607,A -85,B 0,C 180,E1 -7911.229,E2 -7911.229} C_VEL
LIN {X 0,Y 460.677,Z 248.598,A -85,B 0,C 180,E1 -7913.875,E2 -7913.875} C_VEL
LIN {X 0,Y 460.778,Z 248.584,A -85,B 0,C 180,E1 -7917.383,E2 -7917.383} C_VEL
LIN {X 0,Y 460.809,Z 248.584,A -85,B 0,C 180,E1 -7920.005,E2 -7920.005} C_VEL
LIN {X 0,Y 460.749,Z 248.591,A -85,B 0,C 180,E1 -7922.628,E2 -7922.628} C_VEL
LIN {X 0,Y 460.663,Z 248.607,A -85,B 0,C 180,E1 -7926.135,E2 -7926.135} C_VEL
LIN {X 0,Y 460.606,Z 248.606,A -85,B 0,C 180,E1 -7928.781,E2 -7928.781} C_VEL
LIN {X 0,Y 460.608,Z 248.608,A -85,B 0,C 180,E1 -7932.339,E2 -7932.339} C_VEL
LIN {X 0,Y 460.558,Z 248.617,A -85,B 0,C 180,E1 -7935.983,E2 -7935.983} C_VEL
LIN {X 0,Y 460.563,Z 248.617,A -85,B 0,C 180,E1 -7939.62,E2 -7939.62} C_VEL
LIN {X 0,Y 460.51,Z 248.618,A -85,B 0,C 180,E1 -7942.433,E2 -7942.433} C_VEL
LIN {X 0,Y 460.539,Z 248.618,A -85,B 0,C 180,E1 -7945.797,E2 -7945.797} C_VEL
LIN {X 0,Y 460.524,Z 248.621,A -85,B 0,C 180,E1 -7949.236,E2 -7949.236} C_VEL
LIN {X 0,Y 460.524,Z 248.616,A -85,B 0,C 180,E1 -7952.289,E2 -7952.289} C_VEL
LIN {X 0,Y 460.511,Z 248.624,A -85,B 0,C 180,E1 -7955.449,E2 -7955.449} C_VEL
LIN {X 0,Y 460.506,Z 248.625,A -85,B 0,C 180,E1 -7958.893,E2 -7958.893} C_VEL
LIN {X 0,Y 460.515,Z 248.624,A -85,B 0,C 180,E1 -7961.601,E2 -7961.601} C_VEL
LIN {X 0,Y 460.509,Z 248.819,A -85,B 0,C 180,E1 -7962.187,E2 -7962.187} C_VEL
LIN {X 0,Y 461.125,Z 252.627,A -85,B 0,C 180,E1 -7965.487,E2 -7965.487} C_VEL
LIN {X 0,Y 461.458,Z 256.128,A -85,B 0,C 180,E1 -7968.272,E2 -7968.272} C_VEL
LIN {X 0,Y 461.384,Z 259.878,A -85,B 0,C 180,E1 -7970.977,E2 -7970.977} C_VEL
LIN {X 0,Y 460.976,Z 265.319,A -85,B 0,C 180,E1 -7974.596,E2 -7974.596} C_VEL
LIN {X 0,Y 460.709,Z 270.346,A -85,B 0,C 180,E1 -7977.73,E2 -7977.73} C_VEL
LIN {X 0,Y 460.441,Z 275.468,A -85,B 0,C 180,E1 -7980.763,E2 -7980.763} C_VEL
LIN {X 0,Y 460.273,Z 280.705,A -85,B 0,C 180,E1 -7983.717,E2 -7983.717} C_VEL
LIN {X 0,Y 460.06,Z 286.002,A -85,B 0,C 180,E1 -7986.598,E2 -7986.598} C_VEL
LIN {X 0,Y 459.954,Z 291.36,A -85,B 0,C 180,E1 -7989.425,E2 -7989.425} C_VEL
LIN {X 0,Y 459.792,Z 296.826,A -85,B 0,C 180,E1 -7992.2,E2 -7992.2} C_VEL
LIN {X 0,Y 459.747,Z 301.321,A -85,B 0,C 180,E1 -7994.384,E2 -7994.384} C_VEL
LIN {X 0,Y 461.63,Z 311.424,A -85,B 0,C 180,E1 -7994.716,E2 -7994.716} C_VEL
LIN {X 0,Y 463.096,Z 320.637,A -85,B 0,C 180,E1 -7995.105,E2 -7995.105} C_VEL
LIN {X 0,Y 462.896,Z 330,A -85,B 0,C 180,E1 -7995.548,E2 -7995.548} C_VEL
LIN {X 0,Y 462.384,Z 340.143,A -85,B 0,C 180,E1 -7996.15,E2 -7996.15} C_VEL
LIN {X 0,Y 461.928,Z 349.142,A -85,B 0,C 180,E1 -7996.808,E2 -7996.808} C_VEL
LIN {X 0,Y 461.671,Z 357.245,A -85,B 0,C 180,E1 -7997.521,E2 -7997.521} C_VEL
LIN {X 0,Y 461.251,Z 365.278,A -85,B 0,C 180,E1 -7998.353,E2 -7998.353} C_VEL
LIN {X 0,Y 460.87,Z 372.501,A -85,B 0,C 180,E1 -7999.234,E2 -7999.234} C_VEL
LIN {X 0,Y 460.556,Z 378.706,A -85,B 0,C 180,E1 -8000.115,E2 -8000.115} C_VEL
LIN {X 0,Y 460.239,Z 385.246,A -85,B 0,C 180,E1 -8001.217,E2 -8001.217} C_VEL
LIN {X 0,Y 459.987,Z 389.748,A -85,B 0,C 180,E1 -8002.096,E2 -8002.096} C_VEL
LIN {X 0,Y 459.801,Z 395.484,A -85,B 0,C 180,E1 -8003.486,E2 -8003.486} C_VEL
LIN {X 0,Y 459.7,Z 399.566,A -85,B 0,C 180,E1 -8004.737,E2 -8004.737} C_VEL
LIN {X 0,Y 459.583,Z 401.929,A -85,B 0,C 180,E1 -8005.615,E2 -8005.615} C_VEL
LIN {X 0,Y 459.594,Z 403.728,A -85,B 0,C 180,E1 -8006.493,E2 -8006.493} C_VEL
LIN {X 0,Y 459.521,Z 406.169,A -85,B 0,C 180,E1 -8008.247,E2 -8008.247} C_VEL
LIN {X 0,Y 459.498,Z 406.756,A -85,B 0,C 180,E1 -8009.124,E2 -8009.124} C_VEL
LIN {X 0,Y 459.498,Z 406.756,A -85,B 0,C 180,E1 -8010.876,E2 -8010.876} C_VEL
LIN {X 0,Y 459.521,Z 406.169,A -85,B 0,C 180,E1 -8011.753,E2 -8011.753} C_VEL
LIN {X 0,Y 459.594,Z 403.728,A -85,B 0,C 180,E1 -8013.507,E2 -8013.507} C_VEL
LIN {X 0,Y 459.637,Z 400.781,A -85,B 0,C 180,E1 -8014.824,E2 -8014.824} C_VEL
LIN {X 0,Y 459.738,Z 396.794,A -85,B 0,C 180,E1 -8016.143,E2 -8016.143} C_VEL
LIN {X 0,Y 459.889,Z 391.664,A -85,B 0,C 180,E1 -8017.463,E2 -8017.463} C_VEL
LIN {X 0,Y 460.177,Z 386.402,A -85,B 0,C 180,E1 -8018.563,E2 -8018.563} C_VEL
LIN {X 0,Y 460.471,Z 380.083,A -85,B 0,C 180,E1 -8019.665,E2 -8019.665} C_VEL
LIN {X 0,Y 460.756,Z 374.128,A -85,B 0,C 180,E1 -8020.547,E2 -8020.547} C_VEL
LIN {X 0,Y 461.123,Z 367.198,A -85,B 0,C 180,E1 -8021.428,E2 -8021.428} C_VEL
LIN {X 0,Y 461.57,Z 359.015,A -85,B 0,C 180,E1 -8022.308,E2 -8022.308} C_VEL
LIN {X 0,Y 461.881,Z 350.702,A -85,B 0,C 180,E1 -8023.064,E2 -8023.064} C_VEL
LIN {X 0,Y 462.332,Z 341.776,A -85,B 0,C 180,E1 -8023.74,E2 -8023.74} C_VEL
LIN {X 0,Y 462.744,Z 332.013,A -85,B 0,C 180,E1 -8024.344,E2 -8024.344} C_VEL
LIN {X 0,Y 463.115,Z 323.217,A -85,B 0,C 180,E1 -8024.781,E2 -8024.781} C_VEL
LIN {X 0,Y 462.726,Z 318.044,A -85,B 0,C 180,E1 -8025.019,E2 -8025.019} C_VEL
LIN {X 0,Y 460.296,Z 304.364,A -85,B 0,C 180,E1 -8025.532,E2 -8025.532} C_VEL
LIN {X 0,Y 459.74,Z 301.135,A -85,B 0,C 180,E1 -8025.629,E2 -8025.629} C_VEL
LIN {X 0,Y 459.857,Z 295.008,A -85,B 0,C 180,E1 -8028.72,E2 -8028.72} C_VEL
LIN {X 0,Y 460.007,Z 289.564,A -85,B 0,C 180,E1 -8031.51,E2 -8031.51} C_VEL
LIN {X 0,Y 460.115,Z 284.212,A -85,B 0,C 180,E1 -8034.356,E2 -8034.356} C_VEL
LIN {X 0,Y 460.352,Z 278.93,A -85,B 0,C 180,E1 -8037.257,E2 -8037.257} C_VEL
LIN {X 0,Y 460.528,Z 273.743,A -85,B 0,C 180,E1 -8040.238,E2 -8040.238} C_VEL
LIN {X 0,Y 460.766,Z 268.638,A -85,B 0,C 180,E1 -8043.305,E2 -8043.305} C_VEL
LIN {X 0,Y 461.073,Z 263.664,A -85,B 0,C 180,E1 -8046.474,E2 -8046.474} C_VEL
LIN {X 0,Y 461.382,Z 259.875,A -85,B 0,C 180,E1 -8049.023,E2 -8049.023} C_VEL
LIN {X 0,Y 461.454,Z 255.667,A -85,B 0,C 180,E1 -8052.076,E2 -8052.076} C_VEL
LIN {X 0,Y 461.142,Z 252.626,A -85,B 0,C 180,E1 -8054.511,E2 -8054.511} C_VEL
LIN {X 0,Y 460.509,Z 248.816,A -85,B 0,C 180,E1 -8057.813,E2 -8057.813} C_VEL
LIN {X 0,Y 460.518,Z 248.623,A -85,B 0,C 180,E1 -8060.132,E2 -8060.132} C_VEL
LIN {X 0,Y 460.477,Z 248.623,A -85,B 0,C 180,E1 -8063.467,E2 -8063.467} C_VEL
LIN {X 0,Y 460.523,Z 248.624,A -85,B 0,C 180,E1 -8066.671,E2 -8066.671} C_VEL
LIN {X 0,Y 460.508,Z 248.618,A -85,B 0,C 180,E1 -8069.756,E2 -8069.756} C_VEL
LIN {X 0,Y 460.495,Z 248.624,A -85,B 0,C 180,E1 -8072.747,E2 -8072.747} C_VEL
LIN {X 0,Y 460.521,Z 248.617,A -85,B 0,C 180,E1 -8075.663,E2 -8075.663} C_VEL
LIN {X 0,Y 460.522,Z 248.621,A -85,B 0,C 180,E1 -8078.575,E2 -8078.575} C_VEL
LIN {X 0,Y 460.583,Z 248.608,A -85,B 0,C 180,E1 -8081.306,E2 -8081.306} C_VEL
LIN {X 0,Y 460.55,Z 248.613,A -85,B 0,C 180,E1 -8084.96,E2 -8084.96} C_VEL
LIN {X 0,Y 460.607,Z 248.607,A -85,B 0,C 180,E1 -8088.555,E2 -8088.555} C_VEL
LIN {X 0,Y 460.606,Z 248.606,A -85,B 0,C 180,E1 -8091.219,E2 -8091.219} C_VEL
LIN {X 0,Y 460.663,Z 248.607,A -85,B 0,C 180,E1 -8093.865,E2 -8093.865} C_VEL
LIN {X 0,Y 460.749,Z 248.591,A -85,B 0,C 180,E1 -8097.372,E2 -8097.372} C_VEL
LIN {X 0,Y 460.809,Z 248.584,A -85,B 0,C 180,E1 -8099.995,E2 -8099.995} C_VEL
LIN {X 0,Y 460.778,Z 248.584,A -85,B 0,C 180,E1 -8102.617,E2 -8102.617} C_VEL
LIN {X 0,Y 460.677,Z 248.598,A -85,B 0,C 180,E1 -8106.125,E2 -8106.125} C_VEL
LIN {X 0,Y 460.603,Z 248.607,A -85,B 0,C 180,E1 -8108.771,E2 -8108.771} C_VEL
LIN {X 0,Y 460.579,Z 248.609,A -85,B 0,C 180,E1 -8112.43,E2 -8112.43} C_VEL
LIN {X 0,Y 460.58,Z 248.609,A -85,B 0,C 180,E1 -8115.992,E2 -8115.992} C_VEL
LIN {X 0,Y 460.543,Z 248.615,A -85,B 0,C 180,E1 -8119.61,E2 -8119.61} C_VEL
LIN {X 0,Y 460.483,Z 248.622,A -85,B 0,C 180,E1 -8122.423,E2 -8122.423} C_VEL
LIN {X 0,Y 460.524,Z 248.616,A -85,B 0,C 180,E1 -8125.793,E2 -8125.793} C_VEL
LIN {X 0,Y 460.52,Z 248.617,A -85,B 0,C 180,E1 -8128.227,E2 -8128.227} C_VEL
LIN {X 0,Y 460.485,Z 248.622,A -85,B 0,C 180,E1 -8131.277,E2 -8131.277} C_VEL
LIN {X 0,Y 460.496,Z 248.625,A -85,B 0,C 180,E1 -8134.5,E2 -8134.5} C_VEL
LIN {X 0,Y 460.461,Z 248.624,A -85,B 0,C 180,E1 -8137.618,E2 -8137.618} C_VEL
LIN {X 0,Y 460.496,Z 248.624,A -85,B 0,C 180,E1 -8140.264,E2 -8140.264} C_VEL
LIN {X 0,Y 460.479,Z 248.621,A -85,B 0,C 180,E1 -8143.368,E2 -8143.368} C_VEL
LIN {X 0,Y 460.476,Z 248.625,A -85,B 0,C 180,E1 -8146.623,E2 -8146.623} C_VEL
LIN {X 0,Y 460.509,Z 248.62,A -85,B 0,C 180,E1 -8149.723,E2 -8149.723} C_VEL
LIN {X 0,Y 460.475,Z 248.625,A -85,B 0,C 180,E1 -8152.515,E2 -8152.515} C_VEL
LIN {X 0,Y 460.493,Z 248.623,A -85,B 0,C 180,E1 -8155.62,E2 -8155.62} C_VEL
LIN {X 0,Y 460.48,Z 248.622,A -85,B 0,C 180,E1 -8158.741,E2 -8158.741} C_VEL
LIN {X 0,Y 460.499,Z 248.626,A -85,B 0,C 180,E1 -8161.764,E2 -8161.764} C_VEL
LIN {X 0,Y 460.525,Z 248.616,A -85,B 0,C 180,E1 -8164.704,E2 -8164.704} C_VEL
LIN {X 0,Y 460.479,Z 248.628,A -85,B 0,C 180,E1 -8167.57,E2 -8167.57} C_VEL
LIN {X 0,Y 460.507,Z 248.619,A -85,B 0,C 180,E1 -8170.382,E2 -8170.382} C_VEL
LIN {X 0,Y 460.511,Z 248.624,A -85,B 0,C 180,E1 -8173.144,E2 -8173.144} C_VEL
LIN {X 0,Y 460.507,Z 248.623,A -85,B 0,C 180,E1 -8175.867,E2 -8175.867} C_VEL
LIN {X 0,Y 460.571,Z 248.613,A -85,B 0,C 180,E1 -8178.558,E2 -8178.558} C_VEL
LIN {X 0,Y 460.53,Z 248.619,A -85,B 0,C 180,E1 -8179.187,E2 -8179.187} C_VEL
LIN {X 0,Y 459.867,Z 248.706,A -85,B 0,C 180,E1 -8179.917,E2 -8179.917} C_VEL
LIN {X 0,Y 457.049,Z 249.061,A -85,B 0,C 180,E1 -8181.104,E2 -8181.104} C_VEL
LIN {X 0,Y 454.674,Z 249.355,A -85,B 0,C 180,E1 -8182.061,E2 -8182.061} C_VEL
LIN {X 0,Y 453.663,Z 249.477,A -85,B 0,C 180,E1 -8182.799,E2 -8182.799} C_VEL
LIN {X 0,Y 453.585,Z 249.485,A -85,B 0,C 180,E1 -8183.05,E2 -8183.05} C_VEL
LIN {X 0,Y 453.616,Z 249.481,A -85,B 0,C 180,E1 -8184.666,E2 -8184.666} C_VEL
LIN {X 0,Y 453.707,Z 249.472,A -85,B 0,C 180,E1 -8187.337,E2 -8187.337} C_VEL
LIN {X 0,Y 453.755,Z 249.463,A -85,B 0,C 180,E1 -8190,E2 -8190} C_VEL
LIN {X 0,Y 453.707,Z 249.472,A -85,B 0,C 180,E1 -8192.663,E2 -8192.663} C_VEL
LIN {X 0,Y 453.628,Z 249.48,A -85,B 0,C 180,E1 -8196.226,E2 -8196.226} C_VEL
LIN {X 0,Y 453.553,Z 249.491,A -85,B 0,C 180,E1 -8198.914,E2 -8198.914} C_VEL
LIN {X 0,Y 453.536,Z 249.493,A -85,B 0,C 180,E1 -8202.552,E2 -8202.552} C_VEL
LIN {X 0,Y 453.493,Z 249.498,A -85,B 0,C 180,E1 -8206.197,E2 -8206.197} C_VEL
LIN {X 0,Y 453.46,Z 249.499,A -85,B 0,C 180,E1 -8209.044,E2 -8209.044} C_VEL
LIN {X 0,Y 453.443,Z 249.5,A -85,B 0,C 180,E1 -8211.837,E2 -8211.837} C_VEL
LIN {X 0,Y 453.472,Z 249.496,A -85,B 0,C 180,E1 -8214.736,E2 -8214.736} C_VEL
LIN {X 0,Y 453.479,Z 249.499,A -85,B 0,C 180,E1 -8217.964,E2 -8217.964} C_VEL
LIN {X 0,Y 453.427,Z 249.501,A -85,B 0,C 180,E1 -8220.763,E2 -8220.763} C_VEL
LIN {X 0,Y 453.422,Z 249.507,A -85,B 0,C 180,E1 -8223.917,E2 -8223.917} C_VEL
LIN {X 0,Y 453.418,Z 249.502,A -85,B 0,C 180,E1 -8227.192,E2 -8227.192} C_VEL
LIN {X 0,Y 453.481,Z 249.496,A -85,B 0,C 180,E1 -8229.45,E2 -8229.45} C_VEL
LIN {X 0,Y 453.443,Z 249.498,A -85,B 0,C 180,E1 -8232.996,E2 -8232.996} C_VEL
LIN {X 0,Y 453.43,Z 249.505,A -85,B 0,C 180,E1 -8235.785,E2 -8235.785} C_VEL
LIN {X 0,Y 453.449,Z 249.498,A -85,B 0,C 180,E1 -8238.216,E2 -8238.216} C_VEL
LIN {X 0,Y 453.429,Z 249.5,A -85,B 0,C 180,E1 -8240.802,E2 -8240.802} C_VEL
LIN {X 0,Y 453.417,Z 249.503,A -85,B 0,C 180,E1 -8243.923,E2 -8243.923} C_VEL
LIN {X 0,Y 453.446,Z 249.503,A -85,B 0,C 180,E1 -8247.157,E2 -8247.157} C_VEL
LIN {X 0,Y 453.441,Z 249.498,A -85,B 0,C 180,E1 -8250.274,E2 -8250.274} C_VEL
LIN {X 0,Y 453.473,Z 249.499,A -85,B 0,C 180,E1 -8253.299,E2 -8253.299} C_VEL
LIN {X 0,Y 453.472,Z 249.495,A -85,B 0,C 180,E1 -8256.244,E2 -8256.244} C_VEL
LIN {X 0,Y 453.456,Z 249.502,A -85,B 0,C 180,E1 -8259.123,E2 -8259.123} C_VEL
LIN {X 0,Y 453.478,Z 249.494,A -85,B 0,C 180,E1 -8261.95,E2 -8261.95} C_VEL
LIN {X 0,Y 453.515,Z 249.496,A -85,B 0,C 180,E1 -8264.732,E2 -8264.732} C_VEL
LIN {X 0,Y 453.541,Z 249.49,A -85,B 0,C 180,E1 -8268.384,E2 -8268.384} C_VEL
LIN {X 0,Y 453.569,Z 249.484,A -85,B 0,C 180,E1 -8271.092,E2 -8271.092} C_VEL
LIN {X 0,Y 453.645,Z 249.473,A -85,B 0,C 180,E1 -8273.78,E2 -8273.78} C_VEL
LIN {X 0,Y 453.722,Z 249.463,A -85,B 0,C 180,E1 -8277.342,E2 -8277.342} C_VEL
LIN {X 0,Y 453.758,Z 249.462,A -85,B 0,C 180,E1 -8280.005,E2 -8280.005} C_VEL
LIN {X 0,Y 453.696,Z 249.469,A -85,B 0,C 180,E1 -8282.669,E2 -8282.669} C_VEL
LIN {X 0,Y 453.631,Z 249.481,A -85,B 0,C 180,E1 -8286.231,E2 -8286.231} C_VEL
LIN {X 0,Y 453.573,Z 249.482,A -85,B 0,C 180,E1 -8288.918,E2 -8288.918} C_VEL
LIN {X 0,Y 453.564,Z 249.484,A -85,B 0,C 180,E1 -8292.533,E2 -8292.533} C_VEL
LIN {X 0,Y 453.5,Z 249.495,A -85,B 0,C 180,E1 -8296.093,E2 -8296.093} C_VEL
LIN {X 0,Y 453.52,Z 249.489,A -85,B 0,C 180,E1 -8299.043,E2 -8299.043} C_VEL
LIN {X 0,Y 453.478,Z 249.499,A -85,B 0,C 180,E1 -8301.84,E2 -8301.84} C_VEL
LIN {X 0,Y 453.473,Z 249.494,A -85,B 0,C 180,E1 -8304.741,E2 -8304.741} C_VEL
LIN {X 0,Y 453.467,Z 249.497,A -85,B 0,C 180,E1 -8307.946,E2 -8307.946} C_VEL
LIN {X 0,Y 453.463,Z 249.496,A -85,B 0,C 180,E1 -8310.764,E2 -8310.764} C_VEL
LIN {X 0,Y 453.473,Z 249.498,A -85,B 0,C 180,E1 -8313.917,E2 -8313.917} C_VEL
LIN {X 0,Y 453.454,Z 249.504,A -85,B 0,C 180,E1 -8317.193,E2 -8317.193} C_VEL
LIN {X 0,Y 453.479,Z 249.5,A -85,B 0,C 180,E1 -8320.614,E2 -8320.614} C_VEL
LIN {X 0,Y 453.485,Z 249.786,A -85,B 0,C 180,E1 -8321.937,E2 -8321.937} C_VEL
LIN {X 0,Y 454.113,Z 253.678,A -85,B 0,C 180,E1 -8325.394,E2 -8325.394} C_VEL
LIN {X 0,Y 454.46,Z 257.329,A -85,B 0,C 180,E1 -8328.321,E2 -8328.321} C_VEL
LIN {X 0,Y 454.394,Z 260.514,A -85,B 0,C 180,E1 -8330.658,E2 -8330.658} C_VEL
LIN {X 0,Y 454,Z 265.347,A -85,B 0,C 180,E1 -8333.968,E2 -8333.968} C_VEL
LIN {X 0,Y 453.704,Z 270.35,A -85,B 0,C 180,E1 -8337.17,E2 -8337.17} C_VEL
LIN {X 0,Y 453.441,Z 275.437,A -85,B 0,C 180,E1 -8340.266,E2 -8340.266} C_VEL
LIN {X 0,Y 453.237,Z 280.624,A -85,B 0,C 180,E1 -8343.277,E2 -8343.277} C_VEL
LIN {X 0,Y 453.006,Z 285.989,A -85,B 0,C 180,E1 -8346.258,E2 -8346.258} C_VEL
LIN {X 0,Y 452.899,Z 291.236,A -85,B 0,C 180,E1 -8349.09,E2 -8349.09} C_VEL
LIN {X 0,Y 452.711,Z 296.611,A -85,B 0,C 180,E1 -8351.912,E2 -8351.912} C_VEL
LIN {X 0,Y 452.668,Z 300.931,A -85,B 0,C 180,E1 -8354.126,E2 -8354.126} C_VEL
LIN {X 0,Y 454.626,Z 311.701,A -85,B 0,C 180,E1 -8354.491,E2 -8354.491} C_VEL
LIN {X 0,Y 456.041,Z 320.42,A -85,B 0,C 180,E1 -8354.87,E2 -8354.87} C_VEL
LIN {X 0,Y 456.057,Z 328.781,A -85,B 0,C 180,E1 -8355.27,E2 -8355.27} C_VEL
LIN {X 0,Y 455.573,Z 338.299,A -85,B 0,C 180,E1 -8355.824,E2 -8355.824} C_VEL
LIN {X 0,Y 455.087,Z 347.579,A -85,B 0,C 180,E1 -8356.492,E2 -8356.492} C_VEL
LIN {X 0,Y 454.702,Z 357.213,A -85,B 0,C 180,E1 -8357.344,E2 -8357.344} C_VEL
LIN {X 0,Y 454.263,Z 365.066,A -85,B 0,C 180,E1 -8358.171,E2 -8358.171} C_VEL
LIN {X 0,Y 453.866,Z 372.289,A -85,B 0,C 180,E1 -8359.066,E2 -8359.066} C_VEL
LIN {X 0,Y 453.536,Z 378.494,A -85,B 0,C 180,E1 -8359.961,E2 -8359.961} C_VEL
LIN {X 0,Y 453.201,Z 385.034,A -85,B 0,C 180,E1 -8361.079,E2 -8361.079} C_VEL
LIN {X 0,Y 452.931,Z 389.536,A -85,B 0,C 180,E1 -8361.973,E2 -8361.973} C_VEL
LIN {X 0,Y 452.75,Z 394.601,A -85,B 0,C 180,E1 -8363.191,E2 -8363.191} C_VEL
LIN {X 0,Y 452.619,Z 399.354,A -85,B 0,C 180,E1 -8364.654,E2 -8364.654} C_VEL
LIN {X 0,Y 452.505,Z 401.718,A -85,B 0,C 180,E1 -8365.546,E2 -8365.546} C_VEL
LIN {X 0,Y 452.492,Z 403.516,A -85,B 0,C 180,E1 -8366.438,E2 -8366.438} C_VEL
LIN {X 0,Y 452.437,Z 405.958,A -85,B 0,C 180,E1 -8368.22,E2 -8368.22} C_VEL
LIN {X 0,Y 452.407,Z 406.545,A -85,B 0,C 180,E1 -8369.11,E2 -8369.11} C_VEL
LIN {X 0,Y 452.407,Z 406.545,A -85,B 0,C 180,E1 -8370.89,E2 -8370.89} C_VEL
LIN {X 0,Y 452.437,Z 405.958,A -85,B 0,C 180,E1 -8371.78,E2 -8371.78} C_VEL
LIN {X 0,Y 452.492,Z 403.516,A -85,B 0,C 180,E1 -8373.562,E2 -8373.562} C_VEL
LIN {X 0,Y 452.569,Z 400.57,A -85,B 0,C 180,E1 -8374.9,E2 -8374.9} C_VEL
LIN {X 0,Y 452.664,Z 396.582,A -85,B 0,C 180,E1 -8376.239,E2 -8376.239} C_VEL
LIN {X 0,Y 452.837,Z 391.452,A -85,B 0,C 180,E1 -8377.58,E2 -8377.58} C_VEL
LIN {X 0,Y 453.119,Z 386.19,A -85,B 0,C 180,E1 -8378.698,E2 -8378.698} C_VEL
LIN {X 0,Y 453.457,Z 379.871,A -85,B 0,C 180,E1 -8379.816,E2 -8379.816} C_VEL
LIN {X 0,Y 453.736,Z 373.916,A -85,B 0,C 180,E1 -8380.712,E2 -8380.712} C_VEL
LIN {X 0,Y 454.138,Z 366.986,A -85,B 0,C 180,E1 -8381.606,E2 -8381.606} C_VEL
LIN {X 0,Y 454.593,Z 358.802,A -85,B 0,C 180,E1 -8382.5,E2 -8382.5} C_VEL
LIN {X 0,Y 454.951,Z 350.285,A -85,B 0,C 180,E1 -8383.284,E2 -8383.284} C_VEL
LIN {X 0,Y 455.416,Z 341.564,A -85,B 0,C 180,E1 -8383.953,E2 -8383.953} C_VEL
LIN {X 0,Y 455.879,Z 331.802,A -85,B 0,C 180,E1 -8384.565,E2 -8384.565} C_VEL
LIN {X 0,Y 456.238,Z 323.005,A -85,B 0,C 180,E1 -8385.009,E2 -8385.009} C_VEL
LIN {X 0,Y 454.923,Z 313.295,A -85,B 0,C 180,E1 -8385.446,E2 -8385.446} C_VEL
LIN {X 0,Y 452.912,Z 302.678,A -85,B 0,C 180,E1 -8385.823,E2 -8385.823} C_VEL
LIN {X 0,Y 452.664,Z 300.939,A -85,B 0,C 180,E1 -8385.87,E2 -8385.87} C_VEL
LIN {X 0,Y 452.777,Z 294.811,A -85,B 0,C 180,E1 -8389.023,E2 -8389.023} C_VEL
LIN {X 0,Y 452.943,Z 289.439,A -85,B 0,C 180,E1 -8391.863,E2 -8391.863} C_VEL
LIN {X 0,Y 453.079,Z 284.118,A -85,B 0,C 180,E1 -8394.759,E2 -8394.759} C_VEL
LIN {X 0,Y 453.328,Z 278.55,A -85,B 0,C 180,E1 -8397.906,E2 -8397.906} C_VEL
LIN {X 0,Y 453.527,Z 273.712,A -85,B 0,C 180,E1 -8400.755,E2 -8400.755} C_VEL
LIN {X 0,Y 453.778,Z 268.643,A -85,B 0,C 180,E1 -8403.886,E2 -8403.886} C_VEL
LIN {X 0,Y 454.112,Z 263.701,A -85,B 0,C 180,E1 -8407.126,E2 -8407.126} C_VEL
LIN {X 0,Y 454.371,Z 260.474,A -85,B 0,C 180,E1 -8409.357,E2 -8409.357} C_VEL
LIN {X 0,Y 454.468,Z 256.817,A -85,B 0,C 180,E1 -8412.07,E2 -8412.07} C_VEL
LIN {X 0,Y 454.127,Z 253.673,A -85,B 0,C 180,E1 -8414.607,E2 -8414.607} C_VEL
LIN {X 0,Y 453.485,Z 249.785,A -85,B 0,C 180,E1 -8418.063,E2 -8418.063} C_VEL
LIN {X 0,Y 453.45,Z 249.503,A -85,B 0,C 180,E1 -8420.542,E2 -8420.542} C_VEL
LIN {X 0,Y 453.456,Z 249.497,A -85,B 0,C 180,E1 -8423.913,E2 -8423.913} C_VEL
LIN {X 0,Y 453.48,Z 249.495,A -85,B 0,C 180,E1 -8427.147,E2 -8427.147} C_VEL
LIN {X 0,Y 453.466,Z 249.499,A -85,B 0,C 180,E1 -8430.264,E2 -8430.264} C_VEL
LIN {X 0,Y 453.446,Z 249.498,A -85,B 0,C 180,E1 -8433.286,E2 -8433.286} C_VEL
LIN {X 0,Y 453.496,Z 249.497,A -85,B 0,C 180,E1 -8436.234,E2 -8436.234} C_VEL
LIN {X 0,Y 453.477,Z 249.494,A -85,B 0,C 180,E1 -8439.113,E2 -8439.113} C_VEL
LIN {X 0,Y 453.485,Z 249.497,A -85,B 0,C 180,E1 -8441.939,E2 -8441.939} C_VEL
LIN {X 0,Y 453.52,Z 249.49,A -85,B 0,C 180,E1 -8444.721,E2 -8444.721} C_VEL
LIN {X 0,Y 453.556,Z 249.487,A -85,B 0,C 180,E1 -8448.374,E2 -8448.374} C_VEL
LIN {X 0,Y 453.573,Z 249.482,A -85,B 0,C 180,E1 -8451.082,E2 -8451.082} C_VEL
LIN {X 0,Y 453.631,Z 249.481,A -85,B 0,C 180,E1 -8453.769,E2 -8453.769} C_VEL
LIN {X 0,Y 453.696,Z 249.469,A -85,B 0,C 180,E1 -8457.331,E2 -8457.331} C_VEL
LIN {X 0,Y 453.758,Z 249.462,A -85,B 0,C 180,E1 -8459.995,E2 -8459.995} C_VEL
LIN {X 0,Y 453.722,Z 249.463,A -85,B 0,C 180,E1 -8462.658,E2 -8462.658} C_VEL
LIN {X 0,Y 453.645,Z 249.473,A -85,B 0,C 180,E1 -8466.22,E2 -8466.22} C_VEL
LIN {X 0,Y 453.569,Z 249.484,A -85,B 0,C 180,E1 -8468.908,E2 -8468.908} C_VEL
LIN {X 0,Y 453.546,Z 249.485,A -85,B 0,C 180,E1 -8472.523,E2 -8472.523} C_VEL
LIN {X 0,Y 453.524,Z 249.488,A -85,B 0,C 180,E1 -8476.19,E2 -8476.19} C_VEL
LIN {X 0,Y 453.493,Z 249.498,A -85,B 0,C 180,E1 -8479.033,E2 -8479.033} C_VEL
LIN {X 0,Y 453.45,Z 249.497,A -85,B 0,C 180,E1 -8481.83,E2 -8481.83} C_VEL
LIN {X 0,Y 453.475,Z 249.499,A -85,B 0,C 180,E1 -8484.729,E2 -8484.729} C_VEL
LIN {X 0,Y 453.501,Z 249.491,A -85,B 0,C 180,E1 -8487.954,E2 -8487.954} C_VEL
LIN {X 0,Y 453.43,Z 249.5,A -85,B 0,C 180,E1 -8491.519,E2 -8491.519} C_VEL
LIN {X 0,Y 453.451,Z 249.503,A -85,B 0,C 180,E1 -8494.772,E2 -8494.772} C_VEL
LIN {X 0,Y 453.419,Z 249.506,A -85,B 0,C 180,E1 -8498.307,E2 -8498.307} C_VEL
LIN {X 0,Y 453.451,Z 249.503,A -85,B 0,C 180,E1 -8500.604,E2 -8500.604} C_VEL
LIN {X 0,Y 453.436,Z 249.499,A -85,B 0,C 180,E1 -8503.243,E2 -8503.243} C_VEL
LIN {X 0,Y 453.429,Z 249.501,A -85,B 0,C 180,E1 -8505.775,E2 -8505.775} C_VEL
LIN {X 0,Y 453.447,Z 249.505,A -85,B 0,C 180,E1 -8508.207,E2 -8508.207} C_VEL
LIN {X 0,Y 453.48,Z 249.494,A -85,B 0,C 180,E1 -8510.783,E2 -8510.783} C_VEL
LIN {X 0,Y 453.402,Z 249.509,A -85,B 0,C 180,E1 -8513.913,E2 -8513.913} C_VEL
LIN {X 0,Y 453.427,Z 249.5,A -85,B 0,C 180,E1 -8517.147,E2 -8517.147} C_VEL
LIN {X 0,Y 453.456,Z 249.499,A -85,B 0,C 180,E1 -8520.268,E2 -8520.268} C_VEL
LIN {X 0,Y 453.456,Z 249.498,A -85,B 0,C 180,E1 -8523.291,E2 -8523.291} C_VEL
LIN {X 0,Y 453.459,Z 249.498,A -85,B 0,C 180,E1 -8526.237,E2 -8526.237} C_VEL
LIN {X 0,Y 453.455,Z 249.498,A -85,B 0,C 180,E1 -8529.117,E2 -8529.117} C_VEL
LIN {X 0,Y 453.457,Z 249.502,A -85,B 0,C 180,E1 -8531.943,E2 -8531.943} C_VEL
LIN {X 0,Y 453.501,Z 249.495,A -85,B 0,C 180,E1 -8534.725,E2 -8534.725} C_VEL
LIN {X 0,Y 453.523,Z 249.491,A -85,B 0,C 180,E1 -8538.378,E2 -8538.378} C_VEL
LIN {X 0,Y 453.591,Z 249.484,A -85,B 0,C 180,E1 -8541.984,E2 -8541.984} C_VEL
LIN {X 0,Y 453.585,Z 249.485,A -85,B 0,C 180,E1 -8543.05,E2 -8543.05} C_VEL
LIN {X 0,Y 452.9,Z 249.571,A -85,B 0,C 180,E1 -8543.79,E2 -8543.79} C_VEL
LIN {X 0,Y 449.953,Z 249.94,A -85,B 0,C 180,E1 -8544.992,E2 -8544.992} C_VEL
LIN {X 0,Y 447.528,Z 250.24,A -85,B 0,C 180,E1 -8545.962,E2 -8545.962} C_VEL
LIN {X 0,Y 446.584,Z 250.358,A -85,B 0,C 180,E1 -8546.712,E2 -8546.712} C_VEL
LIN {X 0,Y 446.56,Z 250.36,A -85,B 0,C 180,E1 -8546.966,E2 -8546.966} C_VEL
LIN {X 0,Y 446.726,Z 250.339,A -85,B 0,C 180,E1 -8550,E2 -8550} C_VEL
LIN {X 0,Y 446.652,Z 250.351,A -85,B 0,C 180,E1 -8552.706,E2 -8552.706} C_VEL
LIN {X 0,Y 446.596,Z 250.356,A -85,B 0,C 180,E1 -8556.324,E2 -8556.324} C_VEL
LIN {X 0,Y 446.495,Z 250.369,A -85,B 0,C 180,E1 -8559.056,E2 -8559.056} C_VEL
LIN {X 0,Y 446.471,Z 250.374,A -85,B 0,C 180,E1 -8562.731,E2 -8562.731} C_VEL
LIN {X 0,Y 446.455,Z 250.375,A -85,B 0,C 180,E1 -8566.24,E2 -8566.24} C_VEL
LIN {X 0,Y 446.409,Z 250.375,A -85,B 0,C 180,E1 -8569.306,E2 -8569.306} C_VEL
LIN {X 0,Y 446.383,Z 250.383,A -85,B 0,C 180,E1 -8572.201,E2 -8572.201} C_VEL
LIN {X 0,Y 446.415,Z 250.373,A -85,B 0,C 180,E1 -8575.154,E2 -8575.154} C_VEL
LIN {X 0,Y 446.426,Z 250.38,A -85,B 0,C 180,E1 -8578.182,E2 -8578.182} C_VEL
LIN {X 0,Y 446.375,Z 250.379,A -85,B 0,C 180,E1 -8581.303,E2 -8581.303} C_VEL
LIN {X 0,Y 446.375,Z 250.38,A -85,B 0,C 180,E1 -8584.527,E2 -8584.527} C_VEL
LIN {X 0,Y 446.386,Z 250.382,A -85,B 0,C 180,E1 -8588.087,E2 -8588.087} C_VEL
LIN {X 0,Y 446.397,Z 250.376,A -85,B 0,C 180,E1 -8590.925,E2 -8590.925} C_VEL
LIN {X 0,Y 446.397,Z 250.381,A -85,B 0,C 180,E1 -8593.845,E2 -8593.845} C_VEL
LIN {X 0,Y 446.401,Z 250.375,A -85,B 0,C 180,E1 -8596.402,E2 -8596.402} C_VEL
LIN {X 0,Y 446.394,Z 250.38,A -85,B 0,C 180,E1 -8599.807,E2 -8599.807} C_VEL
LIN {X 0,Y 446.363,Z 250.386,A -85,B 0,C 180,E1 -8603.26,E2 -8603.26} C_VEL
LIN {X 0,Y 446.412,Z 250.374,A -85,B 0,C 180,E1 -8606.572,E2 -8606.572} C_VEL
LIN {X 0,Y 446.397,Z 250.376,A -85,B 0,C 180,E1 -8609.985,E2 -8609.985} C_VEL
LIN {X 0,Y 446.442,Z 250.374,A -85,B 0,C 180,E1 -8612.845,E2 -8612.845} C_VEL
LIN {X 0,Y 446.435,Z 250.371,A -85,B 0,C 180,E1 -8615.93,E2 -8615.93} C_VEL
LIN {X 0,Y 446.427,Z 250.377,A -85,B 0,C 180,E1 -8618.779,E2 -8618.779} C_VEL
LIN {X 0,Y 446.427,Z 250.372,A -85,B 0,C 180,E1 -8621.655,E2 -8621.655} C_VEL
LIN {X 0,Y 446.484,Z 250.369,A -85,B 0,C 180,E1 -8624.485,E2 -8624.485} C_VEL
LIN {X 0,Y 446.499,Z 250.365,A -85,B 0,C 180,E1 -8628.199,E2 -8628.199} C_VEL
LIN {X 0,Y 446.516,Z 250.364,A -85,B 0,C 180,E1 -8630.95,E2 -8630.95} C_VEL
LIN {X 0,Y 446.614,Z 250.349,A -85,B 0,C 180,E1 -8633.682,E2 -8633.682} C_VEL
LIN {X 0,Y 446.669,Z 250.342,A -85,B 0,C 180,E1 -8637.3,E2 -8637.3} C_VEL
LIN {X 0,Y 446.709,Z 250.341,A -85,B 0,C 180,E1 -8640.005,E2 -8640.005} C_VEL
LIN {X 0,Y 446.646,Z 250.347,A -85,B 0,C 180,E1 -8642.711,E2 -8642.711} C_VEL
